LIN {X 0,Y 474.723,Z 291.355,A -85,B 0,C 180,E1 -7371.486,E2 -7371.486} C_VEL
LIN {X 0,Y 474.771,Z 291.342,A -85,B 0,C 180,E1 -7374.052,E2 -7374.052} C_VEL
LIN {X 0,Y 474.888,Z 291.331,A -85,B 0,C 180,E1 -7377.455,E2 -7377.455} C_VEL
LIN {X 0,Y 474.905,Z 291.328,A -85,B 0,C 180,E1 -7380,E2 -7380} C_VEL
LIN {X 0,Y 474.888,Z 291.326,A -85,B 0,C 180,E1 -7382.544,E2 -7382.544} C_VEL
LIN {X 0,Y 474.754,Z 291.35,A -85,B 0,C 180,E1 -7385.948,E2 -7385.948} C_VEL
LIN {X 0,Y 474.722,Z 291.348,A -85,B 0,C 180,E1 -7388.513,E2 -7388.513} C_VEL
LIN {X 0,Y 474.699,Z 291.357,A -85,B 0,C 180,E1 -7391.962,E2 -7391.962} C_VEL
LIN {X 0,Y 474.693,Z 291.35,A -85,B 0,C 180,E1 -7395.456,E2 -7395.456} C_VEL
LIN {X 0,Y 474.657,Z 291.355,A -85,B 0,C 180,E1 -7399.01,E2 -7399.01} C_VEL
LIN {X 0,Y 474.582,Z 291.365,A -85,B 0,C 180,E1 -7401.729,E2 -7401.729} C_VEL
LIN {X 0,Y 474.635,Z 291.365,A -85,B 0,C 180,E1 -7404.494,E2 -7404.494} C_VEL
LIN {X 0,Y 474.667,Z 291.353,A -85,B 0,C 180,E1 -7407.333,E2 -7407.333} C_VEL
LIN {X 0,Y 474.599,Z 291.366,A -85,B 0,C 180,E1 -7410.23,E2 -7410.23} C_VEL
LIN {X 0,Y 474.637,Z 291.358,A -85,B 0,C 180,E1 -7413.22,E2 -7413.22} C_VEL
LIN {X 0,Y 474.583,Z 291.367,A -85,B 0,C 180,E1 -7416.324,E2 -7416.324} C_VEL
LIN {X 0,Y 474.611,Z 291.36,A -85,B 0,C 180,E1 -7419.646,E2 -7419.646} C_VEL
LIN {X 0,Y 474.619,Z 291.36,A -85,B 0,C 180,E1 -7422.237,E2 -7422.237} C_VEL
LIN {X 0,Y 474.616,Z 291.363,A -85,B 0,C 180,E1 -7425.298,E2 -7425.298} C_VEL
LIN {X 0,Y 474.599,Z 291.362,A -85,B 0,C 180,E1 -7428.213,E2 -7428.213} C_VEL
LIN {X 0,Y 474.605,Z 291.364,A -85,B 0,C 180,E1 -7431.543,E2 -7431.543} C_VEL
LIN {X 0,Y 474.619,Z 291.361,A -85,B 0,C 180,E1 -7434.726,E2 -7434.726} C_VEL
LIN {X 0,Y 474.631,Z 291.36,A -85,B 0,C 180,E1 -7437.788,E2 -7437.788} C_VEL
LIN {X 0,Y 474.598,Z 291.364,A -85,B 0,C 180,E1 -7440.89,E2 -7440.89} C_VEL
LIN {X 0,Y 474.58,Z 291.37,A -85,B 0,C 180,E1 -7443.624,E2 -7443.624} C_VEL
LIN {X 0,Y 474.632,Z 291.357,A -85,B 0,C 180,E1 -7446.642,E2 -7446.642} C_VEL
LIN {X 0,Y 474.65,Z 291.358,A -85,B 0,C 180,E1 -7450.09,E2 -7450.09} C_VEL
LIN {X 0,Y 474.641,Z 291.361,A -85,B 0,C 180,E1 -7451.655,E2 -7451.655} C_VEL
LIN {X 0,Y 473.971,Z 291.446,A -85,B 0,C 180,E1 -7452.364,E2 -7452.364} C_VEL
LIN {X 0,Y 471.125,Z 291.8,A -85,B 0,C 180,E1 -7453.515,E2 -7453.515} C_VEL
LIN {X 0,Y 468.718,Z 292.097,A -85,B 0,C 180,E1 -7454.444,E2 -7454.444} C_VEL
LIN {X 0,Y 467.68,Z 292.225,A -85,B 0,C 180,E1 -7455.161,E2 -7455.161} C_VEL
LIN {X 0,Y 467.593,Z 292.236,A -85,B 0,C 180,E1 -7455.404,E2 -7455.404} C_VEL
LIN {X 0,Y 467.646,Z 292.237,A -85,B 0,C 180,E1 -7457.855,E2 -7457.855} C_VEL
LIN {X 0,Y 467.608,Z 292.446,A -85,B 0,C 180,E1 -7459.391,E2 -7459.391} C_VEL
LIN {X 0,Y 468.582,Z 298.825,A -85,B 0,C 180,E1 -7460.722,E2 -7460.722} C_VEL
LIN {X 0,Y 468.407,Z 309.742,A -85,B 0,C 180,E1 -7462.891,E2 -7462.891} C_VEL
LIN {X 0,Y 468.423,Z 311.097,A -85,B 0,C 180,E1 -7463.12,E2 -7463.12} C_VEL
LIN {X 0,Y 471.229,Z 325.691,A -85,B 0,C 180,E1 -7463.443,E2 -7463.443} C_VEL
LIN {X 0,Y 470.47,Z 418.633,A -85,B 0,C 180,E1 -7464.885,E2 -7464.885} C_VEL
LIN {X 0,Y 470.184,Z 432.296,A -85,B 0,C 180,E1 -7465.285,E2 -7465.285} C_VEL
LIN {X 0,Y 469.932,Z 444.537,A -85,B 0,C 180,E1 -7465.819,E2 -7465.819} C_VEL
LIN {X 0,Y 469.504,Z 455.551,A -85,B 0,C 180,E1 -7466.46,E2 -7466.46} C_VEL
LIN {X 0,Y 468.905,Z 467.03,A -85,B 0,C 180,E1 -7467.316,E2 -7467.316} C_VEL
LIN {X 0,Y 468.348,Z 477.362,A -85,B 0,C 180,E1 -7468.281,E2 -7468.281} C_VEL
LIN {X 0,Y 468.012,Z 486.652,A -85,B 0,C 180,E1 -7469.355,E2 -7469.355} C_VEL
LIN {X 0,Y 467.614,Z 495.635,A -85,B 0,C 180,E1 -7470.646,E2 -7470.646} C_VEL
LIN {X 0,Y 467.235,Z 502.903,A -85,B 0,C 180,E1 -7471.94,E2 -7471.94} C_VEL
LIN {X 0,Y 467.003,Z 509.572,A -85,B 0,C 180,E1 -7473.451,E2 -7473.451} C_VEL
LIN {X 0,Y 466.785,Z 513.994,A -85,B 0,C 180,E1 -7474.75,E2 -7474.75} C_VEL
LIN {X 0,Y 466.802,Z 517.34,A -85,B 0,C 180,E1 -7476.05,E2 -7476.05} C_VEL
LIN {X 0,Y 466.72,Z 519.012,A -85,B 0,C 180,E1 -7476.919,E2 -7476.919} C_VEL
LIN {X 0,Y 466.647,Z 520.285,A -85,B 0,C 180,E1 -7477.79,E2 -7477.79} C_VEL
LIN {X 0,Y 466.607,Z 521.161,A -85,B 0,C 180,E1 -7478.663,E2 -7478.663} C_VEL
LIN {X 0,Y 466.617,Z 521.635,A -85,B 0,C 180,E1 -7480.413,E2 -7480.413} C_VEL
LIN {X 0,Y 466.682,Z 520.881,A -85,B 0,C 180,E1 -7481.8,E2 -7481.8} C_VEL
LIN {X 0,Y 466.617,Z 519.325,A -85,B 0,C 180,E1 -7483.057,E2 -7483.057} C_VEL
LIN {X 0,Y 466.789,Z 516.721,A -85,B 0,C 180,E1 -7484.385,E2 -7484.385} C_VEL
LIN {X 0,Y 466.913,Z 513.055,A -85,B 0,C 180,E1 -7485.72,E2 -7485.72} C_VEL
LIN {X 0,Y 467.082,Z 508.207,A -85,B 0,C 180,E1 -7487.062,E2 -7487.062} C_VEL
LIN {X 0,Y 467.401,Z 502.021,A -85,B 0,C 180,E1 -7488.407,E2 -7488.407} C_VEL
LIN {X 0,Y 467.778,Z 494.252,A -85,B 0,C 180,E1 -7489.758,E2 -7489.758} C_VEL
LIN {X 0,Y 468.18,Z 486.207,A -85,B 0,C 180,E1 -7490.887,E2 -7490.887} C_VEL
LIN {X 0,Y 468.699,Z 476.286,A -85,B 0,C 180,E1 -7492.016,E2 -7492.016} C_VEL
LIN {X 0,Y 469.231,Z 465.174,A -85,B 0,C 180,E1 -7493.035,E2 -7493.035} C_VEL
LIN {X 0,Y 469.751,Z 454.217,A -85,B 0,C 180,E1 -7493.825,E2 -7493.825} C_VEL
LIN {X 0,Y 470.136,Z 442.648,A -85,B 0,C 180,E1 -7494.477,E2 -7494.477} C_VEL
LIN {X 0,Y 470.465,Z 429.508,A -85,B 0,C 180,E1 -7495.021,E2 -7495.021} C_VEL
LIN {X 0,Y 470.663,Z 418.167,A -85,B 0,C 180,E1 -7495.334,E2 -7495.334} C_VEL
LIN {X 0,Y 471.539,Z 325.876,A -85,B 0,C 180,E1 -7496.773,E2 -7496.773} C_VEL
LIN {X 0,Y 468.472,Z 310.826,A -85,B 0,C 180,E1 -7497.149,E2 -7497.149} C_VEL
LIN {X 0,Y 468.698,Z 298.454,A -85,B 0,C 180,E1 -7499.577,E2 -7499.577} C_VEL
LIN {X 0,Y 467.588,Z 292.242,A -85,B 0,C 180,E1 -7500.909,E2 -7500.909} C_VEL
LIN {X 0,Y 467.588,Z 292.243,A -85,B 0,C 180,E1 -7504.242,E2 -7504.242} C_VEL
LIN {X 0,Y 467.547,Z 292.238,A -85,B 0,C 180,E1 -7507.186,E2 -7507.186} C_VEL
LIN {X 0,Y 467.574,Z 292.243,A -85,B 0,C 180,E1 -7510.265,E2 -7510.265} C_VEL
LIN {X 0,Y 467.586,Z 292.242,A -85,B 0,C 180,E1 -7512.567,E2 -7512.567} C_VEL
LIN {X 0,Y 467.565,Z 292.243,A -85,B 0,C 180,E1 -7515.053,E2 -7515.053} C_VEL
LIN {X 0,Y 467.588,Z 292.236,A -85,B 0,C 180,E1 -7517.44,E2 -7517.44} C_VEL
LIN {X 0,Y 467.581,Z 292.243,A -85,B 0,C 180,E1 -7520.855,E2 -7520.855} C_VEL
LIN {X 0,Y 467.559,Z 292.238,A -85,B 0,C 180,E1 -7524.261,E2 -7524.261} C_VEL
LIN {X 0,Y 467.581,Z 292.238,A -85,B 0,C 180,E1 -7527.321,E2 -7527.321} C_VEL
LIN {X 0,Y 467.569,Z 292.237,A -85,B 0,C 180,E1 -7530.668,E2 -7530.668} C_VEL
LIN {X 0,Y 467.615,Z 292.234,A -85,B 0,C 180,E1 -7533.2,E2 -7533.2} C_VEL
LIN {X 0,Y 467.591,Z 292.23,A -85,B 0,C 180,E1 -7536.468,E2 -7536.468} C_VEL
LIN {X 0,Y 467.621,Z 292.23,A -85,B 0,C 180,E1 -7539.777,E2 -7539.777} C_VEL
LIN {X 0,Y 467.606,Z 292.233,A -85,B 0,C 180,E1 -7542.507,E2 -7542.507} C_VEL
LIN {X 0,Y 467.605,Z 292.233,A -85,B 0,C 180,E1 -7545.197,E2 -7545.197} C_VEL
LIN {X 0,Y 467.655,Z 292.23,A -85,B 0,C 180,E1 -7547.855,E2 -7547.855} C_VEL
LIN {X 0,Y 467.681,Z 292.227,A -85,B 0,C 180,E1 -7551.357,E2 -7551.357} C_VEL
LIN {X 0,Y 467.733,Z 292.222,A -85,B 0,C 180,E1 -7553.963,E2 -7553.963} C_VEL
LIN {X 0,Y 467.859,Z 292.202,A -85,B 0,C 180,E1 -7557.417,E2 -7557.417} C_VEL
LIN {X 0,Y 467.881,Z 292.205,A -85,B 0,C 180,E1 -7560,E2 -7560} C_VEL
LIN {X 0,Y 467.858,Z 292.201,A -85,B 0,C 180,E1 -7562.583,E2 -7562.583} C_VEL
LIN {X 0,Y 467.734,Z 292.222,A -85,B 0,C 180,E1 -7566.038,E2 -7566.038} C_VEL
LIN {X 0,Y 467.681,Z 292.227,A -85,B 0,C 180,E1 -7568.643,E2 -7568.643} C_VEL
LIN {X 0,Y 467.656,Z 292.227,A -85,B 0,C 180,E1 -7572.146,E2 -7572.146} C_VEL
LIN {X 0,Y 467.639,Z 292.226,A -85,B 0,C 180,E1 -7575.695,E2 -7575.695} C_VEL
LIN {X 0,Y 467.617,Z 292.236,A -85,B 0,C 180,E1 -7578.765,E2 -7578.765} C_VEL
LIN {X 0,Y 467.58,Z 292.237,A -85,B 0,C 180,E1 -7581.268,E2 -7581.268} C_VEL
LIN {X 0,Y 467.572,Z 292.236,A -85,B 0,C 180,E1 -7583.944,E2 -7583.944} C_VEL
LIN {X 0,Y 467.617,Z 292.24,A -85,B 0,C 180,E1 -7586.8,E2 -7586.8} C_VEL
LIN {X 0,Y 467.554,Z 292.24,A -85,B 0,C 180,E1 -7589.738,E2 -7589.738} C_VEL
LIN {X 0,Y 467.584,Z 292.239,A -85,B 0,C 180,E1 -7592.759,E2 -7592.759} C_VEL
LIN {X 0,Y 467.554,Z 292.238,A -85,B 0,C 180,E1 -7595.89,E2 -7595.89} C_VEL
LIN {X 0,Y 467.577,Z 292.238,A -85,B 0,C 180,E1 -7599.146,E2 -7599.146} C_VEL
LIN {X 0,Y 467.588,Z 292.235,A -85,B 0,C 180,E1 -7602.567,E2 -7602.567} C_VEL
LIN {X 0,Y 467.567,Z 292.241,A -85,B 0,C 180,E1 -7605.053,E2 -7605.053} C_VEL
LIN {X 0,Y 467.591,Z 292.242,A -85,B 0,C 180,E1 -7607.44,E2 -7607.44} C_VEL
LIN {X 0,Y 467.562,Z 292.24,A -85,B 0,C 180,E1 -7610.853,E2 -7610.853} C_VEL
LIN {X 0,Y 467.562,Z 292.242,A -85,B 0,C 180,E1 -7614.261,E2 -7614.261} C_VEL
LIN {X 0,Y 467.584,Z 292.241,A -85,B 0,C 180,E1 -7617.321,E2 -7617.321} C_VEL
LIN {X 0,Y 467.572,Z 292.241,A -85,B 0,C 180,E1 -7620.668,E2 -7620.668} C_VEL
LIN {X 0,Y 467.656,Z 292.33,A -85,B 0,C 180,E1 -7623.803,E2 -7623.803} C_VEL
LIN {X 0,Y 469.784,Z 303.007,A -85,B 0,C 180,E1 -7625.863,E2 -7625.863} C_VEL
LIN {X 0,Y 469.808,Z 309.972,A -85,B 0,C 180,E1 -7627.111,E2 -7627.111} C_VEL
LIN {X 0,Y 468.912,Z 329.539,A -85,B 0,C 180,E1 -7630.52,E2 -7630.52} C_VEL
LIN {X 0,Y 468.369,Z 343.57,A -85,B 0,C 180,E1 -7632.905,E2 -7632.905} C_VEL
LIN {X 0,Y 471.319,Z 363.38,A -85,B 0,C 180,E1 -7633.336,E2 -7633.336} C_VEL
LIN {X 0,Y 470.655,Z 451.588,A -85,B 0,C 180,E1 -7634.713,E2 -7634.713} C_VEL
LIN {X 0,Y 470.26,Z 464.156,A -85,B 0,C 180,E1 -7635.06,E2 -7635.06} C_VEL
LIN {X 0,Y 469.811,Z 477.1,A -85,B 0,C 180,E1 -7635.599,E2 -7635.599} C_VEL
LIN {X 0,Y 469.33,Z 488.59,A -85,B 0,C 180,E1 -7636.248,E2 -7636.248} C_VEL
LIN {X 0,Y 468.867,Z 499.09,A -85,B 0,C 180,E1 -7637.006,E2 -7637.006} C_VEL
LIN {X 0,Y 468.361,Z 509.888,A -85,B 0,C 180,E1 -7637.983,E2 -7637.983} C_VEL
LIN {X 0,Y 467.794,Z 520.504,A -85,B 0,C 180,E1 -7639.176,E2 -7639.176} C_VEL
LIN {X 0,Y 467.345,Z 529.701,A -85,B 0,C 180,E1 -7640.478,E2 -7640.478} C_VEL
LIN {X 0,Y 467.066,Z 537.117,A -85,B 0,C 180,E1 -7641.781,E2 -7641.781} C_VEL
LIN {X 0,Y 466.851,Z 543.077,A -85,B 0,C 180,E1 -7643.083,E2 -7643.083} C_VEL
LIN {X 0,Y 466.761,Z 547.79,A -85,B 0,C 180,E1 -7644.383,E2 -7644.383} C_VEL
LIN {X 0,Y 466.647,Z 551.39,A -85,B 0,C 180,E1 -7645.681,E2 -7645.681} C_VEL
LIN {X 0,Y 466.69,Z 553.248,A -85,B 0,C 180,E1 -7646.546,E2 -7646.546} C_VEL
LIN {X 0,Y 466.662,Z 554.64,A -85,B 0,C 180,E1 -7647.41,E2 -7647.41} C_VEL
LIN {X 0,Y 466.619,Z 556.241,A -85,B 0,C 180,E1 -7649.137,E2 -7649.137} C_VEL
LIN {X 0,Y 466.601,Z 556.45,A -85,B 0,C 180,E1 -7650,E2 -7650} C_VEL
LIN {X 0,Y 466.619,Z 556.228,A -85,B 0,C 180,E1 -7650.863,E2 -7650.863} C_VEL
LIN {X 0,Y 466.662,Z 554.614,A -85,B 0,C 180,E1 -7652.589,E2 -7652.589} C_VEL
LIN {X 0,Y 466.69,Z 553.205,A -85,B 0,C 180,E1 -7653.453,E2 -7653.453} C_VEL
LIN {X 0,Y 466.689,Z 550.247,A -85,B 0,C 180,E1 -7654.751,E2 -7654.751} C_VEL
LIN {X 0,Y 466.75,Z 546.241,A -85,B 0,C 180,E1 -7656.05,E2 -7656.05} C_VEL
LIN {X 0,Y 466.925,Z 540.074,A -85,B 0,C 180,E1 -7657.568,E2 -7657.568} C_VEL
LIN {X 0,Y 467.165,Z 533.341,A -85,B 0,C 180,E1 -7658.87,E2 -7658.87} C_VEL
LIN {X 0,Y 467.506,Z 524.984,A -85,B 0,C 180,E1 -7660.174,E2 -7660.174} C_VEL
LIN {X 0,Y 467.972,Z 516.394,A -85,B 0,C 180,E1 -7661.258,E2 -7661.258} C_VEL
LIN {X 0,Y 468.463,Z 506.224,A -85,B 0,C 180,E1 -7662.302,E2 -7662.302} C_VEL
LIN {X 0,Y 468.881,Z 495.252,A -85,B 0,C 180,E1 -7663.213,E2 -7663.213} C_VEL
LIN {X 0,Y 469.403,Z 483.651,A -85,B 0,C 180,E1 -7663.97,E2 -7663.97} C_VEL
LIN {X 0,Y 469.866,Z 471.593,A -85,B 0,C 180,E1 -7664.564,E2 -7664.564} C_VEL
LIN {X 0,Y 470.219,Z 458.518,A -85,B 0,C 180,E1 -7665.024,E2 -7665.024} C_VEL
LIN {X 0,Y 470.502,Z 446.174,A -85,B 0,C 180,E1 -7665.291,E2 -7665.291} C_VEL
LIN {X 0,Y 471.087,Z 362.941,A -85,B 0,C 180,E1 -7666.562,E2 -7666.562} C_VEL
LIN {X 0,Y 468.226,Z 343.525,A -85,B 0,C 180,E1 -7666.969,E2 -7666.969} C_VEL
LIN {X 0,Y 468.921,Z 326.108,A -85,B 0,C 180,E1 -7669.935,E2 -7669.935} C_VEL
LIN {X 0,Y 469.726,Z 306.247,A -85,B 0,C 180,E1 -7673.358,E2 -7673.358} C_VEL
LIN {X 0,Y 469.556,Z 302.21,A -85,B 0,C 180,E1 -7674.075,E2 -7674.075} C_VEL
LIN {X 0,Y 467.65,Z 292.236,A -85,B 0,C 180,E1 -7675.957,E2 -7675.957} C_VEL
LIN {X 0,Y 467.577,Z 292.241,A -85,B 0,C 180,E1 -7678.749,E2 -7678.749} C_VEL
LIN {X 0,Y 467.583,Z 292.239,A -85,B 0,C 180,E1 -7681.739,E2 -7681.739} C_VEL
LIN {X 0,Y 467.563,Z 292.239,A -85,B 0,C 180,E1 -7684.832,E2 -7684.832} C_VEL
LIN {X 0,Y 467.564,Z 292.243,A -85,B 0,C 180,E1 -7688.044,E2 -7688.044} C_VEL
LIN {X 0,Y 467.577,Z 292.236,A -85,B 0,C 180,E1 -7691.276,E2 -7691.276} C_VEL
LIN {X 0,Y 467.55,Z 292.241,A -85,B 0,C 180,E1 -7693.82,E2 -7693.82} C_VEL
LIN {X 0,Y 467.552,Z 292.244,A -85,B 0,C 180,E1 -7696.255,E2 -7696.255} C_VEL
LIN {X 0,Y 467.576,Z 292.243,A -85,B 0,C 180,E1 -7698.723,E2 -7698.723} C_VEL
LIN {X 0,Y 467.562,Z 292.239,A -85,B 0,C 180,E1 -7701.955,E2 -7701.955} C_VEL
LIN {X 0,Y 467.561,Z 292.242,A -85,B 0,C 180,E1 -7705.167,E2 -7705.167} C_VEL
LIN {X 0,Y 467.579,Z 292.237,A -85,B 0,C 180,E1 -7708.259,E2 -7708.259} C_VEL
LIN {X 0,Y 467.573,Z 292.241,A -85,B 0,C 180,E1 -7711.25,E2 -7711.25} C_VEL
LIN {X 0,Y 467.606,Z 292.233,A -85,B 0,C 180,E1 -7714.16,E2 -7714.16} C_VEL
LIN {X 0,Y 467.573,Z 292.244,A -85,B 0,C 180,E1 -7716.995,E2 -7716.995} C_VEL
LIN {X 0,Y 467.618,Z 292.232,A -85,B 0,C 180,E1 -7719.777,E2 -7719.777} C_VEL
LIN {X 0,Y 467.604,Z 292.233,A -85,B 0,C 180,E1 -7722.506,E2 -7722.506} C_VEL
LIN {X 0,Y 467.605,Z 292.24,A -85,B 0,C 180,E1 -7725.196,E2 -7725.196} C_VEL
LIN {X 0,Y 467.651,Z 292.23,A -85,B 0,C 180,E1 -7727.854,E2 -7727.854} C_VEL
LIN {X 0,Y 467.677,Z 292.231,A -85,B 0,C 180,E1 -7731.357,E2 -7731.357} C_VEL
LIN {X 0,Y 467.735,Z 292.22,A -85,B 0,C 180,E1 -7733.962,E2 -7733.962} C_VEL
LIN {X 0,Y 467.853,Z 292.207,A -85,B 0,C 180,E1 -7737.417,E2 -7737.417} C_VEL
LIN {X 0,Y 467.875,Z 292.204,A -85,B 0,C 180,E1 -7740,E2 -7740} C_VEL
LIN {X 0,Y 467.854,Z 292.202,A -85,B 0,C 180,E1 -7742.583,E2 -7742.583} C_VEL
LIN {X 0,Y 467.716,Z 292.226,A -85,B 0,C 180,E1 -7746.038,E2 -7746.038} C_VEL
LIN {X 0,Y 467.676,Z 292.225,A -85,B 0,C 180,E1 -7748.643,E2 -7748.643} C_VEL
LIN {X 0,Y 467.65,Z 292.235,A -85,B 0,C 180,E1 -7752.145,E2 -7752.145} C_VEL
LIN {X 0,Y 467.633,Z 292.232,A -85,B 0,C 180,E1 -7755.695,E2 -7755.695} C_VEL
LIN {X 0,Y 467.616,Z 292.231,A -85,B 0,C 180,E1 -7759.308,E2 -7759.308} C_VEL
LIN {X 0,Y 467.529,Z 292.247,A -85,B 0,C 180,E1 -7762.074,E2 -7762.074} C_VEL
LIN {X 0,Y 467.58,Z 292.238,A -85,B 0,C 180,E1 -7764.889,E2 -7764.889} C_VEL
LIN {X 0,Y 467.61,Z 292.233,A -85,B 0,C 180,E1 -7767.77,E2 -7767.77} C_VEL
LIN {X 0,Y 467.562,Z 292.241,A -85,B 0,C 180,E1 -7771.045,E2 -7771.045} C_VEL
LIN {X 0,Y 467.583,Z 292.239,A -85,B 0,C 180,E1 -7774.242,E2 -7774.242} C_VEL
LIN {X 0,Y 467.542,Z 292.243,A -85,B 0,C 180,E1 -7777.186,E2 -7777.186} C_VEL
LIN {X 0,Y 467.569,Z 292.239,A -85,B 0,C 180,E1 -7780.265,E2 -7780.265} C_VEL
LIN {X 0,Y 467.582,Z 292.24,A -85,B 0,C 180,E1 -7782.567,E2 -7782.567} C_VEL
LIN {X 0,Y 467.566,Z 292.245,A -85,B 0,C 180,E1 -7785.053,E2 -7785.053} C_VEL
LIN {X 0,Y 467.56,Z 292.242,A -85,B 0,C 180,E1 -7788.726,E2 -7788.726} C_VEL
LIN {X 0,Y 467.559,Z 292.239,A -85,B 0,C 180,E1 -7791.956,E2 -7791.956} C_VEL
LIN {X 0,Y 467.555,Z 292.247,A -85,B 0,C 180,E1 -7795.167,E2 -7795.167} C_VEL
LIN {X 0,Y 467.578,Z 292.236,A -85,B 0,C 180,E1 -7798.26,E2 -7798.26} C_VEL
LIN {X 0,Y 467.544,Z 292.247,A -85,B 0,C 180,E1 -7801.249,E2 -7801.249} C_VEL
LIN {X 0,Y 467.573,Z 292.237,A -85,B 0,C 180,E1 -7804.402,E2 -7804.402} C_VEL
LIN {X 0,Y 467.574,Z 292.238,A -85,B 0,C 180,E1 -7806.996,E2 -7806.996} C_VEL
LIN {X 0,Y 467.619,Z 292.238,A -85,B 0,C 180,E1 -7809.778,E2 -7809.778} C_VEL
LIN {X 0,Y 467.589,Z 292.235,A -85,B 0,C 180,E1 -7812.506,E2 -7812.506} C_VEL
LIN {X 0,Y 467.602,Z 292.235,A -85,B 0,C 180,E1 -7815.197,E2 -7815.197} C_VEL
LIN {X 0,Y 467.593,Z 292.236,A -85,B 0,C 180,E1 -7815.404,E2 -7815.404} C_VEL
LIN {X 0,Y 466.917,Z 292.326,A -85,B 0,C 180,E1 -7815.883,E2 -7815.883} C_VEL
LIN {X 0,Y 464.102,Z 292.676,A -85,B 0,C 180,E1 -7816.634,E2 -7816.634} C_VEL
LIN {X 0,Y 461.27,Z 293.03,A -85,B 0,C 180,E1 -7817.393,E2 -7817.393} C_VEL
LIN {X 0,Y 460.588,Z 293.114,A -85,B 0,C 180,E1 -7817.883,E2 -7817.883} C_VEL
LIN {X 0,Y 460.589,Z 293.244,A -85,B 0,C 180,E1 -7819.227,E2 -7819.227} C_VEL
LIN {X 0,Y 461.59,Z 299.658,A -85,B 0,C 180,E1 -7820.58,E2 -7820.58} C_VEL
LIN {X 0,Y 461.453,Z 308.434,A -85,B 0,C 180,E1 -7822.344,E2 -7822.344} C_VEL
LIN {X 0,Y 461.421,Z 311.167,A -85,B 0,C 180,E1 -7822.879,E2 -7822.879} C_VEL
LIN {X 0,Y 464.42,Z 327.318,A -85,B 0,C 180,E1 -7823.238,E2 -7823.238} C_VEL
LIN {X 0,Y 463.599,Z 418.669,A -85,B 0,C 180,E1 -7824.673,E2 -7824.673} C_VEL
LIN {X 0,Y 463.295,Z 432.41,A -85,B 0,C 180,E1 -7825.078,E2 -7825.078} C_VEL
LIN {X 0,Y 463.005,Z 445.221,A -85,B 0,C 180,E1 -7825.648,E2 -7825.648} C_VEL
LIN {X 0,Y 462.512,Z 457.693,A -85,B 0,C 180,E1 -7826.407,E2 -7826.407} C_VEL
LIN {X 0,Y 461.896,Z 468.832,A -85,B 0,C 180,E1 -7827.275,E2 -7827.275} C_VEL
LIN {X 0,Y 461.358,Z 478.868,A -85,B 0,C 180,E1 -7828.254,E2 -7828.254} C_VEL
LIN {X 0,Y 460.975,Z 487.898,A -85,B 0,C 180,E1 -7829.345,E2 -7829.345} C_VEL
LIN {X 0,Y 460.554,Z 496.719,A -85,B 0,C 180,E1 -7830.656,E2 -7830.656} C_VEL
LIN {X 0,Y 460.165,Z 503.844,A -85,B 0,C 180,E1 -7831.97,E2 -7831.97} C_VEL
LIN {X 0,Y 459.964,Z 508.65,A -85,B 0,C 180,E1 -7833.066,E2 -7833.066} C_VEL
LIN {X 0,Y 459.754,Z 513.335,A -85,B 0,C 180,E1 -7834.384,E2 -7834.384} C_VEL
LIN {X 0,Y 459.738,Z 516.914,A -85,B 0,C 180,E1 -7835.703,E2 -7835.703} C_VEL
LIN {X 0,Y 459.625,Z 519.502,A -85,B 0,C 180,E1 -7837.027,E2 -7837.027} C_VEL
LIN {X 0,Y 459.542,Z 520.725,A -85,B 0,C 180,E1 -7837.912,E2 -7837.912} C_VEL
LIN {X 0,Y 459.503,Z 521.51,A -85,B 0,C 180,E1 -7838.798,E2 -7838.798} C_VEL
LIN {X 0,Y 459.536,Z 521.875,A -85,B 0,C 180,E1 -7840.575,E2 -7840.575} C_VEL
LIN {X 0,Y 459.588,Z 521.142,A -85,B 0,C 180,E1 -7841.852,E2 -7841.852} C_VEL
LIN {X 0,Y 459.558,Z 519.362,A -85,B 0,C 180,E1 -7843.262,E2 -7843.262} C_VEL
LIN {X 0,Y 459.721,Z 516.652,A -85,B 0,C 180,E1 -7844.611,E2 -7844.611} C_VEL
LIN {X 0,Y 459.879,Z 512.873,A -85,B 0,C 180,E1 -7845.967,E2 -7845.967} C_VEL
LIN {X 0,Y 460.074,Z 507.903,A -85,B 0,C 180,E1 -7847.33,E2 -7847.33} C_VEL
LIN {X 0,Y 460.429,Z 501.585,A -85,B 0,C 180,E1 -7848.696,E2 -7848.696} C_VEL
LIN {X 0,Y 460.779,Z 495.065,A -85,B 0,C 180,E1 -7849.838,E2 -7849.838} C_VEL
LIN {X 0,Y 461.194,Z 487.167,A -85,B 0,C 180,E1 -7850.984,E2 -7850.984} C_VEL
LIN {X 0,Y 461.761,Z 477.198,A -85,B 0,C 180,E1 -7852.154,E2 -7852.154} C_VEL
LIN {X 0,Y 462.313,Z 466.507,A -85,B 0,C 180,E1 -7853.163,E2 -7853.163} C_VEL
LIN {X 0,Y 462.865,Z 455.89,A -85,B 0,C 180,E1 -7853.964,E2 -7853.964} C_VEL
LIN {X 0,Y 463.265,Z 444.078,A -85,B 0,C 180,E1 -7854.662,E2 -7854.662} C_VEL
LIN {X 0,Y 463.654,Z 430.754,A -85,B 0,C 180,E1 -7855.234,E2 -7855.234} C_VEL
LIN {X 0,Y 463.868,Z 418.708,A -85,B 0,C 180,E1 -7855.582,E2 -7855.582} C_VEL
LIN {X 0,Y 464.792,Z 326.54,A -85,B 0,C 180,E1 -7857.043,E2 -7857.043} C_VEL
LIN {X 0,Y 461.586,Z 311.005,A -85,B 0,C 180,E1 -7857.455,E2 -7857.455} C_VEL
LIN {X 0,Y 461.827,Z 300.836,A -85,B 0,C 180,E1 -7859.472,E2 -7859.472} C_VEL
LIN {X 0,Y 460.919,Z 294.908,A -85,B 0,C 180,E1 -7860.717,E2 -7860.717} C_VEL
LIN {X 0,Y 460.543,Z 293.12,A -85,B 0,C 180,E1 -7861.127,E2 -7861.127} C_VEL
LIN {X 0,Y 460.531,Z 293.123,A -85,B 0,C 180,E1 -7864.506,E2 -7864.506} C_VEL
LIN {X 0,Y 460.5,Z 293.115,A -85,B 0,C 180,E1 -7867.623,E2 -7867.623} C_VEL
LIN {X 0,Y 460.538,Z 293.119,A -85,B 0,C 180,E1 -7870.269,E2 -7870.269} C_VEL
LIN {X 0,Y 460.497,Z 293.12,A -85,B 0,C 180,E1 -7873.376,E2 -7873.376} C_VEL
LIN {X 0,Y 460.498,Z 293.126,A -85,B 0,C 180,E1 -7876.625,E2 -7876.625} C_VEL
LIN {X 0,Y 460.541,Z 293.113,A -85,B 0,C 180,E1 -7879.731,E2 -7879.731} C_VEL
LIN {X 0,Y 460.498,Z 293.121,A -85,B 0,C 180,E1 -7882.524,E2 -7882.524} C_VEL
LIN {X 0,Y 460.545,Z 293.111,A -85,B 0,C 180,E1 -7885.624,E2 -7885.624} C_VEL
LIN {X 0,Y 460.536,Z 293.115,A -85,B 0,C 180,E1 -7888.745,E2 -7888.745} C_VEL
LIN {X 0,Y 460.58,Z 293.104,A -85,B 0,C 180,E1 -7892.254,E2 -7892.254} C_VEL
LIN {X 0,Y 460.546,Z 293.112,A -85,B 0,C 180,E1 -7894.705,E2 -7894.705} C_VEL
LIN {X 0,Y 460.51,Z 293.121,A -85,B 0,C 180,E1 -7897.571,E2 -7897.571} C_VEL
LIN {X 0,Y 460.568,Z 293.105,A -85,B 0,C 180,E1 -7900.385,E2 -7900.385} C_VEL
LIN {X 0,Y 460.563,Z 293.114,A -85,B 0,C 180,E1 -7903.146,E2 -7903.146} C_VEL
LIN {X 0,Y 460.554,Z 293.117,A -85,B 0,C 180,E1 -7905.868,E2 -7905.868} C_VEL
LIN {X 0,Y 460.61,Z 293.102,A -85,B 0,C 180,E1 -7908.559,E2 -7908.559} C_VEL
LIN {X 0,Y 460.695,Z 293.096,A -85,B 0,C 180,E1 -7912.109,E2 -7912.109} C_VEL
LIN {X 0,Y 460.692,Z 293.093,A -85,B 0,C 180,E1 -7914.748,E2 -7914.748} C_VEL
LIN {X 0,Y 460.8,Z 293.081,A -85,B 0,C 180,E1 -7917.378,E2 -7917.378} C_VEL
LIN {X 0,Y 460.852,Z 293.081,A -85,B 0,C 180,E1 -7920,E2 -7920} C_VEL
LIN {X 0,Y 460.799,Z 293.079,A -85,B 0,C 180,E1 -7922.623,E2 -7922.623} C_VEL
LIN {X 0,Y 460.7,Z 293.098,A -85,B 0,C 180,E1 -7926.13,E2 -7926.13} C_VEL
LIN {X 0,Y 460.628,Z 293.104,A -85,B 0,C 180,E1 -7928.776,E2 -7928.776} C_VEL
LIN {X 0,Y 460.613,Z 293.107,A -85,B 0,C 180,E1 -7932.445,E2 -7932.445} C_VEL
LIN {X 0,Y 460.6,Z 293.105,A -85,B 0,C 180,E1 -7935.998,E2 -7935.998} C_VEL
LIN {X 0,Y 460.571,Z 293.112,A -85,B 0,C 180,E1 -7938.902,E2 -7938.902} C_VEL
LIN {X 0,Y 460.516,Z 293.116,A -85,B 0,C 180,E1 -7941.486,E2 -7941.486} C_VEL
LIN {X 0,Y 460.542,Z 293.115,A -85,B 0,C 180,E1 -7944.333,E2 -7944.333} C_VEL
LIN {X 0,Y 460.573,Z 293.112,A -85,B 0,C 180,E1 -7947.244,E2 -7947.244} C_VEL
LIN {X 0,Y 460.511,Z 293.118,A -85,B 0,C 180,E1 -7950.24,E2 -7950.24} C_VEL
LIN {X 0,Y 460.529,Z 293.12,A -85,B 0,C 180,E1 -7953.325,E2 -7953.325} C_VEL
LIN {X 0,Y 460.477,Z 293.12,A -85,B 0,C 180,E1 -7956.53,E2 -7956.53} C_VEL
LIN {X 0,Y 460.528,Z 293.106,A -85,B 0,C 180,E1 -7959.863,E2 -7959.863} C_VEL
LIN {X 0,Y 460.514,Z 293.119,A -85,B 0,C 180,E1 -7962.901,E2 -7962.901} C_VEL
LIN {X 0,Y 460.508,Z 293.121,A -85,B 0,C 180,E1 -7965.831,E2 -7965.831} C_VEL
LIN {X 0,Y 460.532,Z 293.117,A -85,B 0,C 180,E1 -7968.989,E2 -7968.989} C_VEL
LIN {X 0,Y 460.52,Z 293.12,A -85,B 0,C 180,E1 -7971.266,E2 -7971.266} C_VEL
LIN {X 0,Y 460.512,Z 293.119,A -85,B 0,C 180,E1 -7974.555,E2 -7974.555} C_VEL
LIN {X 0,Y 460.534,Z 293.119,A -85,B 0,C 180,E1 -7977.716,E2 -7977.716} C_VEL
LIN {X 0,Y 460.542,Z 293.117,A -85,B 0,C 180,E1 -7980.769,E2 -7980.769} C_VEL
LIN {X 0,Y 460.623,Z 293.244,A -85,B 0,C 180,E1 -7983.555,E2 -7983.555} C_VEL
LIN {X 0,Y 462.914,Z 304.669,A -85,B 0,C 180,E1 -7985.8,E2 -7985.8} C_VEL
LIN {X 0,Y 462.899,Z 311.186,A -85,B 0,C 180,E1 -7986.986,E2 -7986.986} C_VEL
LIN {X 0,Y 461.933,Z 330.734,A -85,B 0,C 180,E1 -7990.445,E2 -7990.445} C_VEL
LIN {X 0,Y 461.361,Z 343.102,A -85,B 0,C 180,E1 -7992.603,E2 -7992.603} C_VEL
LIN {X 0,Y 464.573,Z 363.589,A -85,B 0,C 180,E1 -7993.069,E2 -7993.069} C_VEL
LIN {X 0,Y 463.847,Z 452.275,A -85,B 0,C 180,E1 -7994.483,E2 -7994.483} C_VEL
LIN {X 0,Y 463.435,Z 464.514,A -85,B 0,C 180,E1 -7994.835,E2 -7994.835} C_VEL
LIN {X 0,Y 462.958,Z 477.288,A -85,B 0,C 180,E1 -7995.382,E2 -7995.382} C_VEL
LIN {X 0,Y 462.451,Z 488.656,A -85,B 0,C 180,E1 -7996.039,E2 -7996.039} C_VEL
LIN {X 0,Y 461.829,Z 500.689,A -85,B 0,C 180,E1 -7996.945,E2 -7996.945} C_VEL
LIN {X 0,Y 461.344,Z 510.89,A -85,B 0,C 180,E1 -7997.909,E2 -7997.909} C_VEL
LIN {X 0,Y 460.798,Z 520.392,A -85,B 0,C 180,E1 -7999.009,E2 -7999.009} C_VEL
LIN {X 0,Y 460.331,Z 529.551,A -85,B 0,C 180,E1 -8000.332,E2 -8000.332} C_VEL
LIN {X 0,Y 460.002,Z 536.941,A -85,B 0,C 180,E1 -8001.654,E2 -8001.654} C_VEL
LIN {X 0,Y 459.77,Z 542.881,A -85,B 0,C 180,E1 -8002.976,E2 -8002.976} C_VEL
LIN {X 0,Y 459.658,Z 547.577,A -85,B 0,C 180,E1 -8004.296,E2 -8004.296} C_VEL
LIN {X 0,Y 459.565,Z 551.163,A -85,B 0,C 180,E1 -8005.614,E2 -8005.614} C_VEL
LIN {X 0,Y 459.585,Z 553.01,A -85,B 0,C 180,E1 -8006.493,E2 -8006.493} C_VEL
LIN {X 0,Y 459.584,Z 554.395,A -85,B 0,C 180,E1 -8007.37,E2 -8007.37} C_VEL
LIN {X 0,Y 459.523,Z 555.985,A -85,B 0,C 180,E1 -8009.123,E2 -8009.123} C_VEL
LIN {X 0,Y 459.532,Z 556.186,A -85,B 0,C 180,E1 -8010,E2 -8010} C_VEL
LIN {X 0,Y 459.552,Z 555.956,A -85,B 0,C 180,E1 -8010.876,E2 -8010.876} C_VEL
LIN {X 0,Y 459.584,Z 554.33,A -85,B 0,C 180,E1 -8012.629,E2 -8012.629} C_VEL
LIN {X 0,Y 459.586,Z 552.91,A -85,B 0,C 180,E1 -8013.507,E2 -8013.507} C_VEL
LIN {X 0,Y 459.617,Z 549.942,A -85,B 0,C 180,E1 -8014.824,E2 -8014.824} C_VEL
LIN {X 0,Y 459.714,Z 544.872,A -85,B 0,C 180,E1 -8016.43,E2 -8016.43} C_VEL
LIN {X 0,Y 459.892,Z 538.713,A -85,B 0,C 180,E1 -8017.905,E2 -8017.905} C_VEL
LIN {X 0,Y 460.187,Z 531.728,A -85,B 0,C 180,E1 -8019.227,E2 -8019.227} C_VEL
LIN {X 0,Y 460.57,Z 522.964,A -85,B 0,C 180,E1 -8020.551,E2 -8020.551} C_VEL
LIN {X 0,Y 461.068,Z 513.99,A -85,B 0,C 180,E1 -8021.652,E2 -8021.652} C_VEL
LIN {X 0,Y 461.58,Z 503.142,A -85,B 0,C 180,E1 -8022.732,E2 -8022.732} C_VEL
LIN {X 0,Y 462.107,Z 491.641,A -85,B 0,C 180,E1 -8023.634,E2 -8023.634} C_VEL
LIN {X 0,Y 462.647,Z 479.007,A -85,B 0,C 180,E1 -8024.403,E2 -8024.403} C_VEL
LIN {X 0,Y 463.144,Z 465.986,A -85,B 0,C 180,E1 -8024.977,E2 -8024.977} C_VEL
LIN {X 0,Y 463.517,Z 453.152,A -85,B 0,C 180,E1 -8025.359,E2 -8025.359} C_VEL
LIN {X 0,Y 463.877,Z 416.778,A -85,B 0,C 180,E1 -8025.951,E2 -8025.951} C_VEL
LIN {X 0,Y 464.092,Z 362.235,A -85,B 0,C 180,E1 -8026.802,E2 -8026.802} C_VEL
LIN {X 0,Y 461.244,Z 343.19,A -85,B 0,C 180,E1 -8027.221,E2 -8027.221} C_VEL
LIN {X 0,Y 461.908,Z 327.003,A -85,B 0,C 180,E1 -8030.019,E2 -8030.019} C_VEL
LIN {X 0,Y 462.735,Z 308.459,A -85,B 0,C 180,E1 -8033.258,E2 -8033.258} C_VEL
LIN {X 0,Y 462.74,Z 304.459,A -85,B 0,C 180,E1 -8033.97,E2 -8033.97} C_VEL
LIN {X 0,Y 460.589,Z 293.115,A -85,B 0,C 180,E1 -8036.136,E2 -8036.136} C_VEL
LIN {X 0,Y 460.54,Z 293.117,A -85,B 0,C 180,E1 -8039.23,E2 -8039.23} C_VEL
LIN {X 0,Y 460.531,Z 293.121,A -85,B 0,C 180,E1 -8042.284,E2 -8042.284} C_VEL
LIN {X 0,Y 460.509,Z 293.117,A -85,B 0,C 180,E1 -8045.445,E2 -8045.445} C_VEL
LIN {X 0,Y 460.533,Z 293.115,A -85,B 0,C 180,E1 -8048.895,E2 -8048.895} C_VEL
LIN {X 0,Y 460.521,Z 293.12,A -85,B 0,C 180,E1 -8052.181,E2 -8052.181} C_VEL
LIN {X 0,Y 460.511,Z 293.116,A -85,B 0,C 180,E1 -8055.41,E2 -8055.41} C_VEL
LIN {X 0,Y 460.53,Z 293.12,A -85,B 0,C 180,E1 -8058.397,E2 -8058.397} C_VEL
LIN {X 0,Y 460.523,Z 293.116,A -85,B 0,C 180,E1 -8061.266,E2 -8061.266} C_VEL
LIN {X 0,Y 460.507,Z 293.123,A -85,B 0,C 180,E1 -8064.554,E2 -8064.554} C_VEL
LIN {X 0,Y 460.528,Z 293.114,A -85,B 0,C 180,E1 -8067.715,E2 -8067.715} C_VEL
LIN {X 0,Y 460.536,Z 293.12,A -85,B 0,C 180,E1 -8070.769,E2 -8070.769} C_VEL
LIN {X 0,Y 460.559,Z 293.111,A -85,B 0,C 180,E1 -8073.734,E2 -8073.734} C_VEL
LIN {X 0,Y 460.542,Z 293.115,A -85,B 0,C 180,E1 -8076.624,E2 -8076.624} C_VEL
LIN {X 0,Y 460.547,Z 293.117,A -85,B 0,C 180,E1 -8079.452,E2 -8079.452} C_VEL
LIN {X 0,Y 460.554,Z 293.111,A -85,B 0,C 180,E1 -8082.23,E2 -8082.23} C_VEL
LIN {X 0,Y 460.563,Z 293.114,A -85,B 0,C 180,E1 -8084.965,E2 -8084.965} C_VEL
LIN {X 0,Y 460.606,Z 293.105,A -85,B 0,C 180,E1 -8088.559,E2 -8088.559} C_VEL
LIN {X 0,Y 460.69,Z 293.096,A -85,B 0,C 180,E1 -8092.108,E2 -8092.108} C_VEL
LIN {X 0,Y 460.69,Z 293.094,A -85,B 0,C 180,E1 -8094.748,E2 -8094.748} C_VEL
LIN {X 0,Y 460.794,Z 293.086,A -85,B 0,C 180,E1 -8097.377,E2 -8097.377} C_VEL
LIN {X 0,Y 460.846,Z 293.079,A -85,B 0,C 180,E1 -8100,E2 -8100} C_VEL
LIN {X 0,Y 460.795,Z 293.081,A -85,B 0,C 180,E1 -8102.622,E2 -8102.622} C_VEL
LIN {X 0,Y 460.68,Z 293.101,A -85,B 0,C 180,E1 -8106.13,E2 -8106.13} C_VEL
LIN {X 0,Y 460.623,Z 293.103,A -85,B 0,C 180,E1 -8108.776,E2 -8108.776} C_VEL
LIN {X 0,Y 460.608,Z 293.108,A -85,B 0,C 180,E1 -8112.445,E2 -8112.445} C_VEL
LIN {X 0,Y 460.595,Z 293.112,A -85,B 0,C 180,E1 -8115.998,E2 -8115.998} C_VEL
LIN {X 0,Y 460.562,Z 293.111,A -85,B 0,C 180,E1 -8119.616,E2 -8119.616} C_VEL
LIN {X 0,Y 460.505,Z 293.125,A -85,B 0,C 180,E1 -8122.429,E2 -8122.429} C_VEL
LIN {X 0,Y 460.543,Z 293.114,A -85,B 0,C 180,E1 -8125.797,E2 -8125.797} C_VEL
LIN {X 0,Y 460.543,Z 293.117,A -85,B 0,C 180,E1 -8128.233,E2 -8128.233} C_VEL
LIN {X 0,Y 460.515,Z 293.117,A -85,B 0,C 180,E1 -8131.283,E2 -8131.283} C_VEL
LIN {X 0,Y 460.526,Z 293.121,A -85,B 0,C 180,E1 -8134.506,E2 -8134.506} C_VEL
LIN {X 0,Y 460.495,Z 293.118,A -85,B 0,C 180,E1 -8137.624,E2 -8137.624} C_VEL
LIN {X 0,Y 460.533,Z 293.115,A -85,B 0,C 180,E1 -8140.269,E2 -8140.269} C_VEL
LIN {X 0,Y 460.493,Z 293.121,A -85,B 0,C 180,E1 -8143.376,E2 -8143.376} C_VEL
LIN {X 0,Y 460.5,Z 293.121,A -85,B 0,C 180,E1 -8146.626,E2 -8146.626} C_VEL
LIN {X 0,Y 460.52,Z 293.116,A -85,B 0,C 180,E1 -8149.734,E2 -8149.734} C_VEL
LIN {X 0,Y 460.495,Z 293.12,A -85,B 0,C 180,E1 -8152.524,E2 -8152.524} C_VEL
LIN {X 0,Y 460.533,Z 293.117,A -85,B 0,C 180,E1 -8155.623,E2 -8155.623} C_VEL
LIN {X 0,Y 460.534,Z 293.115,A -85,B 0,C 180,E1 -8158.745,E2 -8158.745} C_VEL
LIN {X 0,Y 460.506,Z 293.121,A -85,B 0,C 180,E1 -8161.765,E2 -8161.765} C_VEL
LIN {X 0,Y 460.517,Z 293.116,A -85,B 0,C 180,E1 -8164.704,E2 -8164.704} C_VEL
LIN {X 0,Y 460.508,Z 293.126,A -85,B 0,C 180,E1 -8167.572,E2 -8167.572} C_VEL
LIN {X 0,Y 460.565,Z 293.11,A -85,B 0,C 180,E1 -8170.385,E2 -8170.385} C_VEL
LIN {X 0,Y 460.603,Z 293.111,A -85,B 0,C 180,E1 -8174.059,E2 -8174.059} C_VEL
LIN {X 0,Y 460.601,Z 293.114,A -85,B 0,C 180,E1 -8177.666,E2 -8177.666} C_VEL
LIN {X 0,Y 460.588,Z 293.114,A -85,B 0,C 180,E1 -8177.883,E2 -8177.883} C_VEL
LIN {X 0,Y 460.316,Z 293.433,A -85,B 0,C 180,E1 -8178.367,E2 -8178.367} C_VEL
LIN {X 0,Y 459.222,Z 294.886,A -85,B 0,C 180,E1 -8179.066,E2 -8179.066} C_VEL
LIN {X 0,Y 457.716,Z 297.169,A -85,B 0,C 180,E1 -8179.726,E2 -8179.726} C_VEL
LIN {X 0,Y 455.709,Z 301.095,A -85,B 0,C 180,E1 -8180.585,E2 -8180.585} C_VEL
LIN {X 0,Y 454.664,Z 305.401,A -85,B 0,C 180,E1 -8181.441,E2 -8181.441} C_VEL
LIN {X 0,Y 454.455,Z 311.252,A -85,B 0,C 180,E1 -8182.617,E2 -8182.617} C_VEL
LIN {X 0,Y 457.499,Z 327.13,A -85,B 0,C 180,E1 -8182.997,E2 -8182.997} C_VEL
LIN {X 0,Y 456.728,Z 418.589,A -85,B 0,C 180,E1 -8184.454,E2 -8184.454} C_VEL
LIN {X 0,Y 456.437,Z 431.69,A -85,B 0,C 180,E1 -8184.838,E2 -8184.838} C_VEL
LIN {X 0,Y 456.115,Z 444.808,A -85,B 0,C 180,E1 -8185.416,E2 -8185.416} C_VEL
LIN {X 0,Y 455.636,Z 456.675,A -85,B 0,C 180,E1 -8186.131,E2 -8186.131} C_VEL
LIN {X 0,Y 454.999,Z 466.791,A -85,B 0,C 180,E1 -8186.901,E2 -8186.901} C_VEL
LIN {X 0,Y 454.419,Z 477.256,A -85,B 0,C 180,E1 -8187.895,E2 -8187.895} C_VEL
LIN {X 0,Y 454.063,Z 485.797,A -85,B 0,C 180,E1 -8188.892,E2 -8188.892} C_VEL
LIN {X 0,Y 453.669,Z 493.689,A -85,B 0,C 180,E1 -8190,E2 -8190} C_VEL
LIN {X 0,Y 453.249,Z 501.451,A -85,B 0,C 180,E1 -8191.333,E2 -8191.333} C_VEL
LIN {X 0,Y 452.935,Z 507.66,A -85,B 0,C 180,E1 -8192.668,E2 -8192.668} C_VEL
LIN {X 0,Y 452.772,Z 512.602,A -85,B 0,C 180,E1 -8194.006,E2 -8194.006} C_VEL
LIN {X 0,Y 452.663,Z 516.437,A -85,B 0,C 180,E1 -8195.345,E2 -8195.345} C_VEL
LIN {X 0,Y 452.648,Z 518.814,A -85,B 0,C 180,E1 -8196.441,E2 -8196.441} C_VEL
LIN {X 0,Y 452.455,Z 521.133,A -85,B 0,C 180,E1 -8198.036,E2 -8198.036} C_VEL
LIN {X 0,Y 452.383,Z 522.177,A -85,B 0,C 180,E1 -8199.84,E2 -8199.84} C_VEL
LIN {X 0,Y 452.444,Z 522.116,A -85,B 0,C 180,E1 -8200.743,E2 -8200.743} C_VEL
LIN {X 0,Y 452.511,Z 521.396,A -85,B 0,C 180,E1 -8201.914,E2 -8201.914} C_VEL
LIN {X 0,Y 452.482,Z 519.405,A -85,B 0,C 180,E1 -8203.473,E2 -8203.473} C_VEL
LIN {X 0,Y 452.672,Z 516.591,A -85,B 0,C 180,E1 -8204.843,E2 -8204.843} C_VEL
LIN {X 0,Y 452.839,Z 512.701,A -85,B 0,C 180,E1 -8206.222,E2 -8206.222} C_VEL
LIN {X 0,Y 453.088,Z 507.614,A -85,B 0,C 180,E1 -8207.606,E2 -8207.606} C_VEL
LIN {X 0,Y 453.49,Z 500.953,A -85,B 0,C 180,E1 -8209.03,E2 -8209.03} C_VEL
LIN {X 0,Y 453.915,Z 492.955,A -85,B 0,C 180,E1 -8210.388,E2 -8210.388} C_VEL
LIN {X 0,Y 454.457,Z 484.536,A -85,B 0,C 180,E1 -8211.548,E2 -8211.548} C_VEL
LIN {X 0,Y 454.985,Z 475.251,A -85,B 0,C 180,E1 -8212.6,E2 -8212.6} C_VEL
LIN {X 0,Y 455.543,Z 465.178,A -85,B 0,C 180,E1 -8213.528,E2 -8213.528} C_VEL
LIN {X 0,Y 456.113,Z 454.068,A -85,B 0,C 180,E1 -8214.342,E2 -8214.342} C_VEL
LIN {X 0,Y 456.589,Z 441.706,A -85,B 0,C 180,E1 -8215.042,E2 -8215.042} C_VEL
LIN {X 0,Y 456.912,Z 429.699,A -85,B 0,C 180,E1 -8215.541,E2 -8215.541} C_VEL
LIN {X 0,Y 457.135,Z 418.169,A -85,B 0,C 180,E1 -8215.864,E2 -8215.864} C_VEL
LIN {X 0,Y 458.063,Z 327.474,A -85,B 0,C 180,E1 -8217.319,E2 -8217.319} C_VEL
LIN {X 0,Y 454.706,Z 311.295,A -85,B 0,C 180,E1 -8217.75,E2 -8217.75} C_VEL
LIN {X 0,Y 454.9,Z 301.955,A -85,B 0,C 180,E1 -8219.629,E2 -8219.629} C_VEL
LIN {X 0,Y 453.53,Z 294.195,A -85,B 0,C 180,E1 -8221.298,E2 -8221.298} C_VEL
LIN {X 0,Y 453.476,Z 294.001,A -85,B 0,C 180,E1 -8223.913,E2 -8223.913} C_VEL
LIN {X 0,Y 453.451,Z 293.993,A -85,B 0,C 180,E1 -8227.19,E2 -8227.19} C_VEL
LIN {X 0,Y 453.485,Z 293.995,A -85,B 0,C 180,E1 -8229.45,E2 -8229.45} C_VEL
LIN {X 0,Y 453.476,Z 293.996,A -85,B 0,C 180,E1 -8231.935,E2 -8231.935} C_VEL
LIN {X 0,Y 453.483,Z 293.994,A -85,B 0,C 180,E1 -8235.471,E2 -8235.471} C_VEL
LIN {X 0,Y 453.478,Z 293.995,A -85,B 0,C 180,E1 -8238.209,E2 -8238.209} C_VEL
LIN {X 0,Y 453.509,Z 293.995,A -85,B 0,C 180,E1 -8240.791,E2 -8240.791} C_VEL
LIN {X 0,Y 453.453,Z 293.994,A -85,B 0,C 180,E1 -8243.917,E2 -8243.917} C_VEL
LIN {X 0,Y 453.482,Z 293.996,A -85,B 0,C 180,E1 -8247.151,E2 -8247.151} C_VEL
LIN {X 0,Y 453.474,Z 293.99,A -85,B 0,C 180,E1 -8250.268,E2 -8250.268} C_VEL
LIN {X 0,Y 453.503,Z 293.992,A -85,B 0,C 180,E1 -8253.294,E2 -8253.294} C_VEL
LIN {X 0,Y 453.501,Z 293.985,A -85,B 0,C 180,E1 -8256.239,E2 -8256.239} C_VEL
LIN {X 0,Y 453.482,Z 293.996,A -85,B 0,C 180,E1 -8259.118,E2 -8259.118} C_VEL
LIN {X 0,Y 453.51,Z 293.992,A -85,B 0,C 180,E1 -8261.945,E2 -8261.945} C_VEL
LIN {X 0,Y 453.539,Z 293.982,A -85,B 0,C 180,E1 -8264.726,E2 -8264.726} C_VEL
LIN {X 0,Y 453.559,Z 293.981,A -85,B 0,C 180,E1 -8268.379,E2 -8268.379} C_VEL
LIN {X 0,Y 453.651,Z 293.975,A -85,B 0,C 180,E1 -8271.985,E2 -8271.985} C_VEL
LIN {X 0,Y 453.666,Z 293.969,A -85,B 0,C 180,E1 -8274.667,E2 -8274.667} C_VEL
LIN {X 0,Y 453.744,Z 293.96,A -85,B 0,C 180,E1 -8277.337,E2 -8277.337} C_VEL
LIN {X 0,Y 453.822,Z 293.956,A -85,B 0,C 180,E1 -8280,E2 -8280} C_VEL
LIN {X 0,Y 453.743,Z 293.958,A -85,B 0,C 180,E1 -8282.664,E2 -8282.664} C_VEL
LIN {X 0,Y 453.668,Z 293.972,A -85,B 0,C 180,E1 -8286.226,E2 -8286.226} C_VEL
LIN {X 0,Y 453.592,Z 293.979,A -85,B 0,C 180,E1 -8288.914,E2 -8288.914} C_VEL
LIN {X 0,Y 453.563,Z 293.986,A -85,B 0,C 180,E1 -8292.529,E2 -8292.529} C_VEL
LIN {X 0,Y 453.545,Z 293.986,A -85,B 0,C 180,E1 -8296.196,E2 -8296.196} C_VEL
LIN {X 0,Y 453.52,Z 293.989,A -85,B 0,C 180,E1 -8299.041,E2 -8299.041} C_VEL
LIN {X 0,Y 453.477,Z 293.993,A -85,B 0,C 180,E1 -8301.836,E2 -8301.836} C_VEL
LIN {X 0,Y 453.514,Z 293.992,A -85,B 0,C 180,E1 -8304.735,E2 -8304.735} C_VEL
LIN {X 0,Y 453.533,Z 293.985,A -85,B 0,C 180,E1 -8307.96,E2 -8307.96} C_VEL
LIN {X 0,Y 453.466,Z 293.995,A -85,B 0,C 180,E1 -8311.525,E2 -8311.525} C_VEL
LIN {X 0,Y 453.488,Z 293.996,A -85,B 0,C 180,E1 -8314.777,E2 -8314.777} C_VEL
LIN {X 0,Y 453.464,Z 293.994,A -85,B 0,C 180,E1 -8318.312,E2 -8318.312} C_VEL
LIN {X 0,Y 453.495,Z 293.981,A -85,B 0,C 180,E1 -8320.609,E2 -8320.609} C_VEL
LIN {X 0,Y 453.456,Z 294.002,A -85,B 0,C 180,E1 -8323.244,E2 -8323.244} C_VEL
LIN {X 0,Y 453.463,Z 294,A -85,B 0,C 180,E1 -8325.779,E2 -8325.779} C_VEL
LIN {X 0,Y 453.481,Z 293.995,A -85,B 0,C 180,E1 -8328.209,E2 -8328.209} C_VEL
LIN {X 0,Y 453.489,Z 293.993,A -85,B 0,C 180,E1 -8330.795,E2 -8330.795} C_VEL
LIN {X 0,Y 453.456,Z 294.003,A -85,B 0,C 180,E1 -8333.917,E2 -8333.917} C_VEL
LIN {X 0,Y 453.485,Z 293.996,A -85,B 0,C 180,E1 -8337.151,E2 -8337.151} C_VEL
LIN {X 0,Y 453.477,Z 293.999,A -85,B 0,C 180,E1 -8340.268,E2 -8340.268} C_VEL
LIN {X 0,Y 453.579,Z 294.164,A -85,B 0,C 180,E1 -8343.298,E2 -8343.298} C_VEL
LIN {X 0,Y 455.937,Z 305.802,A -85,B 0,C 180,E1 -8345.63,E2 -8345.63} C_VEL
LIN {X 0,Y 456.113,Z 309.808,A -85,B 0,C 180,E1 -8346.383,E2 -8346.383} C_VEL
LIN {X 0,Y 455.136,Z 328.036,A -85,B 0,C 180,E1 -8349.669,E2 -8349.669} C_VEL
LIN {X 0,Y 454.449,Z 342.816,A -85,B 0,C 180,E1 -8352.297,E2 -8352.297} C_VEL
LIN {X 0,Y 457.79,Z 363.659,A -85,B 0,C 180,E1 -8352.787,E2 -8352.787} C_VEL
LIN {X 0,Y 457.076,Z 451.942,A -85,B 0,C 180,E1 -8354.219,E2 -8354.219} C_VEL
LIN {X 0,Y 456.632,Z 464.198,A -85,B 0,C 180,E1 -8354.575,E2 -8354.575} C_VEL
LIN {X 0,Y 456.114,Z 477.54,A -85,B 0,C 180,E1 -8355.157,E2 -8355.157} C_VEL
LIN {X 0,Y 455.565,Z 488.758,A -85,B 0,C 180,E1 -8355.824,E2 -8355.824} C_VEL
LIN {X 0,Y 454.951,Z 500.316,A -85,B 0,C 180,E1 -8356.71,E2 -8356.71} C_VEL
LIN {X 0,Y 454.391,Z 510.853,A -85,B 0,C 180,E1 -8357.721,E2 -8357.721} C_VEL
LIN {X 0,Y 453.815,Z 520.304,A -85,B 0,C 180,E1 -8358.838,E2 -8358.838} C_VEL
LIN {X 0,Y 453.303,Z 529.421,A -85,B 0,C 180,E1 -8360.18,E2 -8360.18} C_VEL
LIN {X 0,Y 452.95,Z 536.784,A -85,B 0,C 180,E1 -8361.523,E2 -8361.523} C_VEL
LIN {X 0,Y 452.716,Z 542.701,A -85,B 0,C 180,E1 -8362.866,E2 -8362.866} C_VEL
LIN {X 0,Y 452.557,Z 547.376,A -85,B 0,C 180,E1 -8364.206,E2 -8364.206} C_VEL
LIN {X 0,Y 452.487,Z 550.946,A -85,B 0,C 180,E1 -8365.546,E2 -8365.546} C_VEL
LIN {X 0,Y 452.482,Z 552.777,A -85,B 0,C 180,E1 -8366.438,E2 -8366.438} C_VEL
LIN {X 0,Y 452.508,Z 554.155,A -85,B 0,C 180,E1 -8367.329,E2 -8367.329} C_VEL
LIN {X 0,Y 452.43,Z 555.73,A -85,B 0,C 180,E1 -8369.11,E2 -8369.11} C_VEL
LIN {X 0,Y 452.465,Z 555.92,A -85,B 0,C 180,E1 -8370,E2 -8370} C_VEL
LIN {X 0,Y 452.457,Z 555.056,A -85,B 0,C 180,E1 -8371.78,E2 -8371.78} C_VEL
LIN {X 0,Y 452.508,Z 554.042,A -85,B 0,C 180,E1 -8372.67,E2 -8372.67} C_VEL
LIN {X 0,Y 452.484,Z 552.607,A -85,B 0,C 180,E1 -8373.562,E2 -8373.562} C_VEL
LIN {X 0,Y 452.545,Z 549.626,A -85,B 0,C 180,E1 -8374.9,E2 -8374.9} C_VEL
LIN {X 0,Y 452.611,Z 545.027,A -85,B 0,C 180,E1 -8376.396,E2 -8376.396} C_VEL
LIN {X 0,Y 452.841,Z 538.352,A -85,B 0,C 180,E1 -8378.029,E2 -8378.029} C_VEL
LIN {X 0,Y 453.128,Z 531.335,A -85,B 0,C 180,E1 -8379.372,E2 -8379.372} C_VEL
LIN {X 0,Y 453.55,Z 522.534,A -85,B 0,C 180,E1 -8380.716,E2 -8380.716} C_VEL
LIN {X 0,Y 454.141,Z 512.539,A -85,B 0,C 180,E1 -8381.945,E2 -8381.945} C_VEL
LIN {X 0,Y 454.606,Z 502.436,A -85,B 0,C 180,E1 -8382.946,E2 -8382.946} C_VEL
LIN {X 0,Y 455.165,Z 491.031,A -85,B 0,C 180,E1 -8383.846,E2 -8383.846} C_VEL
LIN {X 0,Y 455.707,Z 479.303,A -85,B 0,C 180,E1 -8384.57,E2 -8384.57} C_VEL
LIN {X 0,Y 456.192,Z 466.566,A -85,B 0,C 180,E1 -8385.154,E2 -8385.154} C_VEL
LIN {X 0,Y 456.592,Z 454.144,A -85,B 0,C 180,E1 -8385.54,E2 -8385.54} C_VEL
LIN {X 0,Y 456.855,Z 433.65,A -85,B 0,C 180,E1 -8385.903,E2 -8385.903} C_VEL
LIN {X 0,Y 457.311,Z 363.451,A -85,B 0,C 180,E1 -8387.008,E2 -8387.008} C_VEL
LIN {X 0,Y 454.254,Z 343.068,A -85,B 0,C 180,E1 -8387.441,E2 -8387.441} C_VEL
LIN {X 0,Y 455.107,Z 323.917,A -85,B 0,C 180,E1 -8390.804,E2 -8390.804} C_VEL
LIN {X 0,Y 455.873,Z 306.81,A -85,B 0,C 180,E1 -8393.846,E2 -8393.846} C_VEL
LIN {X 0,Y 453.928,Z 295.932,A -85,B 0,C 180,E1 -8395.919,E2 -8395.919} C_VEL
LIN {X 0,Y 453.54,Z 293.991,A -85,B 0,C 180,E1 -8396.322,E2 -8396.322} C_VEL
LIN {X 0,Y 453.51,Z 293.994,A -85,B 0,C 180,E1 -8398.711,E2 -8398.711} C_VEL
LIN {X 0,Y 453.464,Z 293.998,A -85,B 0,C 180,E1 -8401.799,E2 -8401.799} C_VEL
LIN {X 0,Y 453.479,Z 293.993,A -85,B 0,C 180,E1 -8404.989,E2 -8404.989} C_VEL
LIN {X 0,Y 453.459,Z 294.004,A -85,B 0,C 180,E1 -8408.311,E2 -8408.311} C_VEL
LIN {X 0,Y 453.492,Z 293.996,A -85,B 0,C 180,E1 -8410.608,E2 -8410.608} C_VEL
LIN {X 0,Y 453.452,Z 293.996,A -85,B 0,C 180,E1 -8413.243,E2 -8413.243} C_VEL
LIN {X 0,Y 453.461,Z 293.995,A -85,B 0,C 180,E1 -8415.778,E2 -8415.778} C_VEL
LIN {X 0,Y 453.477,Z 293.996,A -85,B 0,C 180,E1 -8418.209,E2 -8418.209} C_VEL
LIN {X 0,Y 453.507,Z 293.996,A -85,B 0,C 180,E1 -8420.79,E2 -8420.79} C_VEL
LIN {X 0,Y 453.451,Z 293.996,A -85,B 0,C 180,E1 -8423.917,E2 -8423.917} C_VEL
LIN {X 0,Y 453.479,Z 293.997,A -85,B 0,C 180,E1 -8427.151,E2 -8427.151} C_VEL
LIN {X 0,Y 453.471,Z 293.994,A -85,B 0,C 180,E1 -8430.268,E2 -8430.268} C_VEL
LIN {X 0,Y 453.503,Z 293.994,A -85,B 0,C 180,E1 -8433.293,E2 -8433.293} C_VEL
LIN {X 0,Y 453.499,Z 293.99,A -85,B 0,C 180,E1 -8436.238,E2 -8436.238} C_VEL
LIN {X 0,Y 453.479,Z 294.001,A -85,B 0,C 180,E1 -8439.117,E2 -8439.117} C_VEL
LIN {X 0,Y 453.507,Z 293.99,A -85,B 0,C 180,E1 -8441.944,E2 -8441.944} C_VEL
LIN {X 0,Y 453.537,Z 293.987,A -85,B 0,C 180,E1 -8444.726,E2 -8444.726} C_VEL
LIN {X 0,Y 453.555,Z 293.983,A -85,B 0,C 180,E1 -8448.379,E2 -8448.379} C_VEL
LIN {X 0,Y 453.647,Z 293.974,A -85,B 0,C 180,E1 -8451.985,E2 -8451.985} C_VEL
LIN {X 0,Y 453.664,Z 293.969,A -85,B 0,C 180,E1 -8454.666,E2 -8454.666} C_VEL
LIN {X 0,Y 453.738,Z 293.964,A -85,B 0,C 180,E1 -8457.336,E2 -8457.336} C_VEL
LIN {X 0,Y 453.816,Z 293.955,A -85,B 0,C 180,E1 -8460,E2 -8460} C_VEL
LIN {X 0,Y 453.739,Z 293.96,A -85,B 0,C 180,E1 -8462.663,E2 -8462.663} C_VEL
LIN {X 0,Y 453.646,Z 293.976,A -85,B 0,C 180,E1 -8466.226,E2 -8466.226} C_VEL
LIN {X 0,Y 453.586,Z 293.979,A -85,B 0,C 180,E1 -8468.913,E2 -8468.913} C_VEL
LIN {X 0,Y 453.558,Z 293.985,A -85,B 0,C 180,E1 -8472.529,E2 -8472.529} C_VEL
LIN {X 0,Y 453.539,Z 293.994,A -85,B 0,C 180,E1 -8476.196,E2 -8476.196} C_VEL
LIN {X 0,Y 453.511,Z 293.989,A -85,B 0,C 180,E1 -8479.039,E2 -8479.039} C_VEL
LIN {X 0,Y 453.471,Z 293.996,A -85,B 0,C 180,E1 -8481.836,E2 -8481.836} C_VEL
LIN {X 0,Y 453.494,Z 293.995,A -85,B 0,C 180,E1 -8484.735,E2 -8484.735} C_VEL
LIN {X 0,Y 453.523,Z 293.989,A -85,B 0,C 180,E1 -8487.959,E2 -8487.959} C_VEL
LIN {X 0,Y 453.46,Z 293.995,A -85,B 0,C 180,E1 -8491.525,E2 -8491.525} C_VEL
LIN {X 0,Y 453.482,Z 293.999,A -85,B 0,C 180,E1 -8494.778,E2 -8494.778} C_VEL
LIN {X 0,Y 453.457,Z 293.998,A -85,B 0,C 180,E1 -8498.312,E2 -8498.312} C_VEL
LIN {X 0,Y 453.489,Z 293.997,A -85,B 0,C 180,E1 -8500.609,E2 -8500.609} C_VEL
LIN {X 0,Y 453.45,Z 294,A -85,B 0,C 180,E1 -8503.244,E2 -8503.244} C_VEL
LIN {X 0,Y 453.457,Z 293.995,A -85,B 0,C 180,E1 -8505.779,E2 -8505.779} C_VEL
LIN {X 0,Y 453.466,Z 293.998,A -85,B 0,C 180,E1 -8509.413,E2 -8509.413} C_VEL
LIN {X 0,Y 453.448,Z 294,A -85,B 0,C 180,E1 -8512.811,E2 -8512.811} C_VEL
LIN {X 0,Y 453.465,Z 293.994,A -85,B 0,C 180,E1 -8516.087,E2 -8516.087} C_VEL
LIN {X 0,Y 453.471,Z 294.001,A -85,B 0,C 180,E1 -8519.241,E2 -8519.241} C_VEL
LIN {X 0,Y 453.472,Z 293.993,A -85,B 0,C 180,E1 -8522.294,E2 -8522.294} C_VEL
LIN {X 0,Y 453.465,Z 293.999,A -85,B 0,C 180,E1 -8525.263,E2 -8525.263} C_VEL
LIN {X 0,Y 453.479,Z 293.993,A -85,B 0,C 180,E1 -8528.416,E2 -8528.416} C_VEL
LIN {X 0,Y 453.521,Z 293.988,A -85,B 0,C 180,E1 -8531.009,E2 -8531.009} C_VEL
LIN {X 0,Y 453.568,Z 293.989,A -85,B 0,C 180,E1 -8533.88,E2 -8533.88} C_VEL
LIN {X 0,Y 453.563,Z 293.988,A -85,B 0,C 180,E1 -8537.472,E2 -8537.472} C_VEL
LIN {X 0,Y 453.551,Z 294.044,A -85,B 0,C 180,E1 -8539.058,E2 -8539.058} C_VEL
LIN {X 0,Y 454.657,Z 301.577,A -85,B 0,C 180,E1 -8540.66,E2 -8540.66} C_VEL
LIN {X 0,Y 454.664,Z 305.401,A -85,B 0,C 180,E1 -8541.441,E2 -8541.441} C_VEL
LIN {X 0,Y 454.408,Z 307.858,A -85,B 0,C 180,E1 -8541.814,E2 -8541.814} C_VEL
LIN {X 0,Y 453.924,Z 310.902,A -85,B 0,C 180,E1 -8542.111,E2 -8542.111} C_VEL
LIN {X 0,Y 452.967,Z 316.141,A -85,B 0,C 180,E1 -8542.432,E2 -8542.432} C_VEL
LIN {X 0,Y 451.933,Z 321.942,A -85,B 0,C 180,E1 -8542.638,E2 -8542.638} C_VEL
LIN {X 0,Y 451.326,Z 325.974,A -85,B 0,C 180,E1 -8542.733,E2 -8542.733} C_VEL
LIN {X 0,Y 450.703,Z 334.167,A -85,B 0,C 180,E1 -8542.872,E2 -8542.872} C_VEL
LIN {X 0,Y 449.839,Z 419.525,A -85,B 0,C 180,E1 -8544.256,E2 -8544.256} C_VEL
LIN {X 0,Y 449.518,Z 433.158,A -85,B 0,C 180,E1 -8544.674,E2 -8544.674} C_VEL
LIN {X 0,Y 449.2,Z 445.399,A -85,B 0,C 180,E1 -8545.233,E2 -8545.233} C_VEL
LIN {X 0,Y 448.703,Z 457.18,A -85,B 0,C 180,E1 -8545.959,E2 -8545.959} C_VEL
LIN {X 0,Y 448.03,Z 467.259,A -85,B 0,C 180,E1 -8546.741,E2 -8546.741} C_VEL
LIN {X 0,Y 447.438,Z 477.691,A -85,B 0,C 180,E1 -8547.75,E2 -8547.75} C_VEL
LIN {X 0,Y 447.022,Z 487.085,A -85,B 0,C 180,E1 -8548.874,E2 -8548.874} C_VEL
LIN {X 0,Y 446.54,Z 496.153,A -85,B 0,C 180,E1 -8550.226,E2 -8550.226} C_VEL
LIN {X 0,Y 446.085,Z 503.477,A -85,B 0,C 180,E1 -8551.58,E2 -8551.58} C_VEL
LIN {X 0,Y 445.828,Z 510.208,A -85,B 0,C 180,E1 -8553.163,E2 -8553.163} C_VEL
LIN {X 0,Y 445.561,Z 514.669,A -85,B 0,C 180,E1 -8554.524,E2 -8554.524} C_VEL
LIN {X 0,Y 445.593,Z 517.013,A -85,B 0,C 180,E1 -8555.43,E2 -8555.43} C_VEL
LIN {X 0,Y 445.576,Z 519.14,A -85,B 0,C 180,E1 -8556.441,E2 -8556.441} C_VEL
LIN {X 0,Y 445.35,Z 521.517,A -85,B 0,C 180,E1 -8558.165,E2 -8558.165} C_VEL
LIN {X 0,Y 445.308,Z 522.466,A -85,B 0,C 180,E1 -8559.998,E2 -8559.998} C_VEL
LIN {X 0,Y 445.356,Z 522.341,A -85,B 0,C 180,E1 -8560.916,E2 -8560.916} C_VEL
LIN {X 0,Y 445.427,Z 521.657,A -85,B 0,C 180,E1 -8561.974,E2 -8561.974} C_VEL
LIN {X 0,Y 445.43,Z 519.454,A -85,B 0,C 180,E1 -8563.69,E2 -8563.69} C_VEL
LIN {X 0,Y 445.635,Z 516.538,A -85,B 0,C 180,E1 -8565.083,E2 -8565.083} C_VEL
LIN {X 0,Y 445.806,Z 512.54,A -85,B 0,C 180,E1 -8566.485,E2 -8566.485} C_VEL
LIN {X 0,Y 446.166,Z 506.297,A -85,B 0,C 180,E1 -8568.126,E2 -8568.126} C_VEL
LIN {X 0,Y 446.613,Z 499.414,A -85,B 0,C 180,E1 -8569.536,E2 -8569.536} C_VEL
LIN {X 0,Y 446.998,Z 492.329,A -85,B 0,C 180,E1 -8570.718,E2 -8570.718} C_VEL
LIN {X 0,Y 447.59,Z 483.734,A -85,B 0,C 180,E1 -8571.896,E2 -8571.896} C_VEL
LIN {X 0,Y 448.172,Z 474.214,A -85,B 0,C 180,E1 -8572.959,E2 -8572.959} C_VEL
LIN {X 0,Y 448.809,Z 463.753,A -85,B 0,C 180,E1 -8573.903,E2 -8573.903} C_VEL
LIN {X 0,Y 449.362,Z 452.735,A -85,B 0,C 180,E1 -8574.698,E2 -8574.698} C_VEL
LIN {X 0,Y 449.863,Z 440.437,A -85,B 0,C 180,E1 -8575.382,E2 -8575.382} C_VEL
LIN {X 0,Y 450.189,Z 427.591,A -85,B 0,C 180,E1 -8575.889,E2 -8575.889} C_VEL
LIN {X 0,Y 450.45,Z 416.053,A -85,B 0,C 180,E1 -8576.184,E2 -8576.184} C_VEL
LIN {X 0,Y 451.404,Z 328.618,A -85,B 0,C 180,E1 -8577.6,E2 -8577.6} C_VEL
LIN {X 0,Y 447.825,Z 311.58,A -85,B 0,C 180,E1 -8578.06,E2 -8578.06} C_VEL
LIN {X 0,Y 447.939,Z 302.699,A -85,B 0,C 180,E1 -8579.877,E2 -8579.877} C_VEL
LIN {X 0,Y 446.458,Z 294.874,A -85,B 0,C 180,E1 -8581.605,E2 -8581.605} C_VEL
LIN {X 0,Y 446.429,Z 294.88,A -85,B 0,C 180,E1 -8584.523,E2 -8584.523} C_VEL
LIN {X 0,Y 446.414,Z 294.872,A -85,B 0,C 180,E1 -8588.079,E2 -8588.079} C_VEL
LIN {X 0,Y 446.426,Z 294.877,A -85,B 0,C 180,E1 -8590.918,E2 -8590.918} C_VEL
LIN {X 0,Y 446.399,Z 294.877,A -85,B 0,C 180,E1 -8593.846,E2 -8593.846} C_VEL
LIN {X 0,Y 446.398,Z 294.881,A -85,B 0,C 180,E1 -8596.403,E2 -8596.403} C_VEL
LIN {X 0,Y 446.426,Z 294.876,A -85,B 0,C 180,E1 -8599.082,E2 -8599.082} C_VEL
LIN {X 0,Y 446.414,Z 294.871,A -85,B 0,C 180,E1 -8601.921,E2 -8601.921} C_VEL
LIN {X 0,Y 446.428,Z 294.871,A -85,B 0,C 180,E1 -8605.477,E2 -8605.477} C_VEL
LIN {X 0,Y 446.415,Z 294.873,A -85,B 0,C 180,E1 -8608.7,E2 -8608.7} C_VEL
LIN {X 0,Y 446.484,Z 294.86,A -85,B 0,C 180,E1 -8611.821,E2 -8611.821} C_VEL
LIN {X 0,Y 446.449,Z 294.869,A -85,B 0,C 180,E1 -8614.847,E2 -8614.847} C_VEL
LIN {X 0,Y 446.447,Z 294.868,A -85,B 0,C 180,E1 -8618.245,E2 -8618.245} C_VEL
LIN {X 0,Y 446.456,Z 294.874,A -85,B 0,C 180,E1 -8621.649,E2 -8621.649} C_VEL
LIN {X 0,Y 446.507,Z 294.858,A -85,B 0,C 180,E1 -8624.48,E2 -8624.48} C_VEL
LIN {X 0,Y 446.517,Z 294.859,A -85,B 0,C 180,E1 -8628.193,E2 -8628.193} C_VEL
LIN {X 0,Y 446.6,Z 294.855,A -85,B 0,C 180,E1 -8631.858,E2 -8631.858} C_VEL
LIN {X 0,Y 446.64,Z 294.845,A -85,B 0,C 180,E1 -8634.583,E2 -8634.583} C_VEL
LIN {X 0,Y 446.664,Z 294.844,A -85,B 0,C 180,E1 -8638.197,E2 -8638.197} C_VEL
LIN {X 0,Y 446.792,Z 294.832,A -85,B 0,C 180,E1 -8640,E2 -8640} C_VEL
LIN {X 0,Y 446.69,Z 294.836,A -85,B 0,C 180,E1 -8642.706,E2 -8642.706} C_VEL
LIN {X 0,Y 446.638,Z 294.846,A -85,B 0,C 180,E1 -8646.324,E2 -8646.324} C_VEL
LIN {X 0,Y 446.537,Z 294.857,A -85,B 0,C 180,E1 -8649.056,E2 -8649.056} C_VEL
LIN {X 0,Y 446.521,Z 294.863,A -85,B 0,C 180,E1 -8652.73,E2 -8652.73} C_VEL
LIN {X 0,Y 446.496,Z 294.864,A -85,B 0,C 180,E1 -8656.228,E2 -8656.228} C_VEL
LIN {X 0,Y 446.469,Z 294.865,A -85,B 0,C 180,E1 -8659.303,E2 -8659.303} C_VEL
LIN {X 0,Y 446.418,Z 294.874,A -85,B 0,C 180,E1 -8662.2,E2 -8662.2} C_VEL
LIN {X 0,Y 446.458,Z 294.871,A -85,B 0,C 180,E1 -8665.153,E2 -8665.153} C_VEL
LIN {X 0,Y 446.485,Z 294.864,A -85,B 0,C 180,E1 -8668.179,E2 -8668.179} C_VEL
LIN {X 0,Y 446.419,Z 294.871,A -85,B 0,C 180,E1 -8671.775,E2 -8671.775} C_VEL
LIN {X 0,Y 446.429,Z 294.873,A -85,B 0,C 180,E1 -8674.523,E2 -8674.523} C_VEL
LIN {X 0,Y 446.415,Z 294.873,A -85,B 0,C 180,E1 -8678.079,E2 -8678.079} C_VEL
LIN {X 0,Y 446.428,Z 294.863,A -85,B 0,C 180,E1 -8680.918,E2 -8680.918} C_VEL
LIN {X 0,Y 446.401,Z 294.876,A -85,B 0,C 180,E1 -8683.846,E2 -8683.846} C_VEL
LIN {X 0,Y 446.397,Z 294.876,A -85,B 0,C 180,E1 -8686.404,E2 -8686.404} C_VEL
LIN {X 0,Y 446.428,Z 294.875,A -85,B 0,C 180,E1 -8689.083,E2 -8689.083} C_VEL
LIN {X 0,Y 446.409,Z 294.874,A -85,B 0,C 180,E1 -8692.121,E2 -8692.121} C_VEL
LIN {X 0,Y 446.431,Z 294.875,A -85,B 0,C 180,E1 -8695.477,E2 -8695.477} C_VEL
LIN {X 0,Y 446.418,Z 294.876,A -85,B 0,C 180,E1 -8698.7,E2 -8698.7} C_VEL
LIN {X 0,Y 446.487,Z 294.87,A -85,B 0,C 180,E1 -8701.821,E2 -8701.821} C_VEL
LIN {X 0,Y 446.523,Z 294.992,A -85,B 0,C 180,E1 -8703.011,E2 -8703.011} C_VEL
LIN {X 0,Y 448.808,Z 305.989,A -85,B 0,C 180,E1 -8705.263,E2 -8705.263} C_VEL
LIN {X 0,Y 449.228,Z 311.049,A -85,B 0,C 180,E1 -8706.243,E2 -8706.243} C_VEL
LIN {X 0,Y 448.276,Z 327.961,A -85,B 0,C 180,E1 -8709.344,E2 -8709.344} C_VEL
LIN {X 0,Y 447.527,Z 342.542,A -85,B 0,C 180,E1 -8711.981,E2 -8711.981} C_VEL
LIN {X 0,Y 451.078,Z 364.464,A -85,B 0,C 180,E1 -8712.509,E2 -8712.509} C_VEL
LIN {X 0,Y 450.323,Z 451.72,A -85,B 0,C 180,E1 -8713.947,E2 -8713.947} C_VEL
LIN {X 0,Y 449.851,Z 463.956,A -85,B 0,C 180,E1 -8714.307,E2 -8714.307} C_VEL
LIN {X 0,Y 449.3,Z 476.724,A -85,B 0,C 180,E1 -8714.869,E2 -8714.869} C_VEL
LIN {X 0,Y 448.673,Z 488.89,A -85,B 0,C 180,E1 -8715.601,E2 -8715.601} C_VEL
LIN {X 0,Y 448.029,Z 500.62,A -85,B 0,C 180,E1 -8716.523,E2 -8716.523} C_VEL
LIN {X 0,Y 447.442,Z 510.844,A -85,B 0,C 180,E1 -8717.527,E2 -8717.527} C_VEL
LIN {X 0,Y 446.842,Z 520.234,A -85,B 0,C 180,E1 -8718.661,E2 -8718.661} C_VEL
LIN {X 0,Y 446.286,Z 529.31,A -85,B 0,C 180,E1 -8720.024,E2 -8720.024} C_VEL
LIN {X 0,Y 445.885,Z 536.642,A -85,B 0,C 180,E1 -8721.388,E2 -8721.388} C_VEL
LIN {X 0,Y 445.633,Z 542.533,A -85,B 0,C 180,E1 -8722.752,E2 -8722.752} C_VEL
LIN {X 0,Y 445.47,Z 546.686,A -85,B 0,C 180,E1 -8723.955,E2 -8723.955} C_VEL
LIN {X 0,Y 445.412,Z 550.737,A -85,B 0,C 180,E1 -8725.475,E2 -8725.475} C_VEL
LIN {X 0,Y 445.38,Z 552.549,A -85,B 0,C 180,E1 -8726.381,E2 -8726.381} C_VEL
LIN {X 0,Y 445.433,Z 553.919,A -85,B 0,C 180,E1 -8727.287,E2 -8727.287} C_VEL
LIN {X 0,Y 445.341,Z 555.478,A -85,B 0,C 180,E1 -8729.095,E2 -8729.095} C_VEL
LIN {X 0,Y 445.371,Z 555.651,A -85,B 0,C 180,E1 -8730,E2 -8730} C_VEL
LIN {X 0,Y 445.374,Z 554.771,A -85,B 0,C 180,E1 -8731.808,E2 -8731.808} C_VEL
LIN {X 0,Y 445.433,Z 553.75,A -85,B 0,C 180,E1 -8732.713,E2 -8732.713} C_VEL
LIN {X 0,Y 445.384,Z 552.296,A -85,B 0,C 180,E1 -8733.618,E2 -8733.618} C_VEL
LIN {X 0,Y 445.474,Z 549.3,A -85,B 0,C 180,E1 -8734.977,E2 -8734.977} C_VEL
LIN {X 0,Y 445.557,Z 543.777,A -85,B 0,C 180,E1 -8736.748,E2 -8736.748} C_VEL
LIN {X 0,Y 445.768,Z 537.976,A -85,B 0,C 180,E1 -8738.157,E2 -8738.157} C_VEL
LIN {X 0,Y 446.071,Z 530.921,A -85,B 0,C 180,E1 -8739.522,E2 -8739.522} C_VEL
LIN {X 0,Y 446.544,Z 522.081,A -85,B 0,C 180,E1 -8740.886,E2 -8740.886} C_VEL
LIN {X 0,Y 447.142,Z 512.041,A -85,B 0,C 180,E1 -8742.135,E2 -8742.135} C_VEL
LIN {X 0,Y 447.621,Z 501.859,A -85,B 0,C 180,E1 -8743.151,E2 -8743.151} C_VEL
LIN {X 0,Y 448.212,Z 490.379,A -85,B 0,C 180,E1 -8744.066,E2 -8744.066} C_VEL
LIN {X 0,Y 448.793,Z 478.548,A -85,B 0,C 180,E1 -8744.8,E2 -8744.8} C_VEL
LIN {X 0,Y 449.351,Z 465.549,A -85,B 0,C 180,E1 -8745.39,E2 -8745.39} C_VEL
LIN {X 0,Y 449.732,Z 452.739,A -85,B 0,C 180,E1 -8745.783,E2 -8745.783} C_VEL
LIN {X 0,Y 450.1,Z 418.569,A -85,B 0,C 180,E1 -8746.359,E2 -8746.359} C_VEL
LIN {X 0,Y 450.446,Z 364.085,A -85,B 0,C 180,E1 -8747.231,E2 -8747.231} C_VEL
LIN {X 0,Y 447.254,Z 342.784,A -85,B 0,C 180,E1 -8747.693,E2 -8747.693} C_VEL
LIN {X 0,Y 448.101,Z 324.781,A -85,B 0,C 180,E1 -8750.904,E2 -8750.904} C_VEL
LIN {X 0,Y 448.88,Z 308.86,A -85,B 0,C 180,E1 -8753.775,E2 -8753.775} C_VEL
LIN {X 0,Y 448.227,Z 303.619,A -85,B 0,C 180,E1 -8754.77,E2 -8754.77} C_VEL
LIN {X 0,Y 446.524,Z 294.863,A -85,B 0,C 180,E1 -8756.512,E2 -8756.512} C_VEL
LIN {X 0,Y 446.449,Z 294.873,A -85,B 0,C 180,E1 -8759.209,E2 -8759.209} C_VEL
LIN {X 0,Y 446.422,Z 294.877,A -85,B 0,C 180,E1 -8762.361,E2 -8762.361} C_VEL
LIN {X 0,Y 446.418,Z 294.873,A -85,B 0,C 180,E1 -8765.625,E2 -8765.625} C_VEL
LIN {X 0,Y 446.436,Z 294.871,A -85,B 0,C 180,E1 -8769.027,E2 -8769.027} C_VEL
LIN {X 0,Y 446.432,Z 294.877,A -85,B 0,C 180,E1 -8772.277,E2 -8772.277} C_VEL
LIN {X 0,Y 446.449,Z 294.87,A -85,B 0,C 180,E1 -8775.103,E2 -8775.103} C_VEL
LIN {X 0,Y 446.426,Z 294.88,A -85,B 0,C 180,E1 -8778.608,E2 -8778.608} C_VEL
LIN {X 0,Y 446.452,Z 294.872,A -85,B 0,C 180,E1 -8780.974,E2 -8780.974} C_VEL
LIN {X 0,Y 446.416,Z 294.876,A -85,B 0,C 180,E1 -8784.373,E2 -8784.373} C_VEL
LIN {X 0,Y 446.418,Z 294.872,A -85,B 0,C 180,E1 -8787.638,E2 -8787.638} C_VEL
LIN {X 0,Y 446.445,Z 294.875,A -85,B 0,C 180,E1 -8790.79,E2 -8790.79} C_VEL
LIN {X 0,Y 446.474,Z 294.865,A -85,B 0,C 180,E1 -8793.848,E2 -8793.848} C_VEL
LIN {X 0,Y 446.425,Z 294.876,A -85,B 0,C 180,E1 -8796.823,E2 -8796.823} C_VEL
LIN {X 0,Y 446.44,Z 294.871,A -85,B 0,C 180,E1 -8799.737,E2 -8799.737} C_VEL
LIN {X 0,Y 446.459,Z 294.868,A -85,B 0,C 180,E1 -8802.597,E2 -8802.597} C_VEL
LIN {X 0,Y 446.467,Z 294.873,A -85,B 0,C 180,E1 -8805.412,E2 -8805.412} C_VEL
LIN {X 0,Y 446.513,Z 294.861,A -85,B 0,C 180,E1 -8808.193,E2 -8808.193} C_VEL
LIN {X 0,Y 446.595,Z 294.854,A -85,B 0,C 180,E1 -8811.858,E2 -8811.858} C_VEL
LIN {X 0,Y 446.638,Z 294.845,A -85,B 0,C 180,E1 -8814.582,E2 -8814.582} C_VEL
LIN {X 0,Y 446.658,Z 294.844,A -85,B 0,C 180,E1 -8818.196,E2 -8818.196} C_VEL
LIN {X 0,Y 446.786,Z 294.831,A -85,B 0,C 180,E1 -8820,E2 -8820} C_VEL
LIN {X 0,Y 446.686,Z 294.839,A -85,B 0,C 180,E1 -8822.705,E2 -8822.705} C_VEL
LIN {X 0,Y 446.614,Z 294.851,A -85,B 0,C 180,E1 -8826.324,E2 -8826.324} C_VEL
LIN {X 0,Y 446.532,Z 294.858,A -85,B 0,C 180,E1 -8829.055,E2 -8829.055} C_VEL
LIN {X 0,Y 446.516,Z 294.861,A -85,B 0,C 180,E1 -8832.73,E2 -8832.73} C_VEL
LIN {X 0,Y 446.49,Z 294.871,A -85,B 0,C 180,E1 -8836.227,E2 -8836.227} C_VEL
LIN {X 0,Y 446.462,Z 294.866,A -85,B 0,C 180,E1 -8839.303,E2 -8839.303} C_VEL
LIN {X 0,Y 446.413,Z 294.879,A -85,B 0,C 180,E1 -8842.2,E2 -8842.2} C_VEL
LIN {X 0,Y 446.436,Z 294.87,A -85,B 0,C 180,E1 -8845.153,E2 -8845.153} C_VEL
LIN {X 0,Y 446.479,Z 294.869,A -85,B 0,C 180,E1 -8848.179,E2 -8848.179} C_VEL
LIN {X 0,Y 446.413,Z 294.873,A -85,B 0,C 180,E1 -8851.775,E2 -8851.775} C_VEL
LIN {X 0,Y 446.424,Z 294.878,A -85,B 0,C 180,E1 -8854.523,E2 -8854.523} C_VEL
LIN {X 0,Y 446.409,Z 294.874,A -85,B 0,C 180,E1 -8858.079,E2 -8858.079} C_VEL
LIN {X 0,Y 446.422,Z 294.879,A -85,B 0,C 180,E1 -8860.918,E2 -8860.918} C_VEL
LIN {X 0,Y 446.396,Z 294.875,A -85,B 0,C 180,E1 -8863.846,E2 -8863.846} C_VEL
LIN {X 0,Y 446.389,Z 294.877,A -85,B 0,C 180,E1 -8866.405,E2 -8866.405} C_VEL
LIN {X 0,Y 446.398,Z 294.875,A -85,B 0,C 180,E1 -8869.798,E2 -8869.798} C_VEL
LIN {X 0,Y 446.402,Z 294.874,A -85,B 0,C 180,E1 -8872.121,E2 -8872.121} C_VEL
LIN {X 0,Y 446.419,Z 294.877,A -85,B 0,C 180,E1 -8875.477,E2 -8875.477} C_VEL
LIN {X 0,Y 446.411,Z 294.874,A -85,B 0,C 180,E1 -8878.7,E2 -8878.7} C_VEL
LIN {X 0,Y 446.421,Z 294.875,A -85,B 0,C 180,E1 -8881.837,E2 -8881.837} C_VEL
LIN {X 0,Y 446.417,Z 294.873,A -85,B 0,C 180,E1 -8884.846,E2 -8884.846} C_VEL
LIN {X 0,Y 446.446,Z 294.87,A -85,B 0,C 180,E1 -8888.246,E2 -8888.246} C_VEL
LIN {X 0,Y 446.447,Z 294.877,A -85,B 0,C 180,E1 -8891.649,E2 -8891.649} C_VEL
LIN {X 0,Y 446.506,Z 294.863,A -85,B 0,C 180,E1 -8894.48,E2 -8894.48} C_VEL
LIN {X 0,Y 446.505,Z 294.869,A -85,B 0,C 180,E1 -8898.193,E2 -8898.193} C_VEL
LIN {X 0,Y 446.537,Z 294.981,A -85,B 0,C 180,E1 -8898.913,E2 -8898.913} C_VEL
LIN {X 0,Y 447.683,Z 302.414,A -85,B 0,C 180,E1 -8900.513,E2 -8900.513} C_VEL
LIN {X 0,Y 447.483,Z 311.532,A -85,B 0,C 180,E1 -8902.379,E2 -8902.379} C_VEL
LIN {X 0,Y 450.707,Z 328.385,A -85,B 0,C 180,E1 -8902.778,E2 -8902.778} C_VEL
LIN {X 0,Y 450.703,Z 334.167,A -85,B 0,C 180,E1 -8902.872,E2 -8902.872} C_VEL
LIN {X 0,Y 450.021,Z 340.008,A -85,B 0,C 180,E1 -8902.943,E2 -8902.943} C_VEL
LIN {X 0,Y 444.309,Z 358.989,A -85,B 0,C 180,E1 -8903.054,E2 -8903.054} C_VEL
LIN {X 0,Y 443.596,Z 364.832,A -85,B 0,C 180,E1 -8903.125,E2 -8903.125} C_VEL
LIN {X 0,Y 442.979,Z 419.241,A -85,B 0,C 180,E1 -8904.024,E2 -8904.024} C_VEL
LIN {X 0,Y 442.664,Z 432.307,A -85,B 0,C 180,E1 -8904.42,E2 -8904.42} C_VEL
LIN {X 0,Y 442.327,Z 444.854,A -85,B 0,C 180,E1 -8904.987,E2 -8904.987} C_VEL
LIN {X 0,Y 441.841,Z 456.082,A -85,B 0,C 180,E1 -8905.667,E2 -8905.667} C_VEL
LIN {X 0,Y 441.174,Z 466.411,A -85,B 0,C 180,E1 -8906.461,E2 -8906.461} C_VEL
LIN {X 0,Y 440.546,Z 477.037,A -85,B 0,C 180,E1 -8907.486,E2 -8907.486} C_VEL
LIN {X 0,Y 440.041,Z 486.599,A -85,B 0,C 180,E1 -8908.628,E2 -8908.628} C_VEL
LIN {X 0,Y 439.628,Z 494.448,A -85,B 0,C 180,E1 -8909.771,E2 -8909.771} C_VEL
LIN {X 0,Y 439.143,Z 502.159,A -85,B 0,C 180,E1 -8911.147,E2 -8911.147} C_VEL
LIN {X 0,Y 438.801,Z 509.229,A -85,B 0,C 180,E1 -8912.754,E2 -8912.754} C_VEL
LIN {X 0,Y 438.574,Z 513.96,A -85,B 0,C 180,E1 -8914.136,E2 -8914.136} C_VEL
LIN {X 0,Y 438.503,Z 517.585,A -85,B 0,C 180,E1 -8915.519,E2 -8915.519} C_VEL
LIN {X 0,Y 438.504,Z 519.461,A -85,B 0,C 180,E1 -8916.442,E2 -8916.442} C_VEL
LIN {X 0,Y 438.328,Z 520.888,A -85,B 0,C 180,E1 -8917.37,E2 -8917.37} C_VEL
LIN {X 0,Y 438.215,Z 522.521,A -85,B 0,C 180,E1 -8919.229,E2 -8919.229} C_VEL
LIN {X 0,Y 438.238,Z 522.749,A -85,B 0,C 180,E1 -8920.161,E2 -8920.161} C_VEL
LIN {X 0,Y 438.269,Z 522.537,A -85,B 0,C 180,E1 -8921.095,E2 -8921.095} C_VEL
LIN {X 0,Y 438.335,Z 521.926,A -85,B 0,C 180,E1 -8922.031,E2 -8922.031} C_VEL
LIN {X 0,Y 438.299,Z 520.92,A -85,B 0,C 180,E1 -8922.973,E2 -8922.973} C_VEL
LIN {X 0,Y 438.38,Z 519.485,A -85,B 0,C 180,E1 -8923.915,E2 -8923.915} C_VEL
LIN {X 0,Y 438.595,Z 516.475,A -85,B 0,C 180,E1 -8925.331,E2 -8925.331} C_VEL
LIN {X 0,Y 438.786,Z 512.358,A -85,B 0,C 180,E1 -8926.757,E2 -8926.757} C_VEL
LIN {X 0,Y 439.2,Z 505.971,A -85,B 0,C 180,E1 -8928.424,E2 -8928.424} C_VEL
LIN {X 0,Y 439.678,Z 498.956,A -85,B 0,C 180,E1 -8929.857,E2 -8929.857} C_VEL
LIN {X 0,Y 440.106,Z 491.72,A -85,B 0,C 180,E1 -8931.057,E2 -8931.057} C_VEL
LIN {X 0,Y 440.798,Z 481.908,A -85,B 0,C 180,E1 -8932.371,E2 -8932.371} C_VEL
LIN {X 0,Y 441.459,Z 471.891,A -85,B 0,C 180,E1 -8933.453,E2 -8933.453} C_VEL
LIN {X 0,Y 442.18,Z 460.853,A -85,B 0,C 180,E1 -8934.409,E2 -8934.409} C_VEL
LIN {X 0,Y 442.78,Z 448.902,A -85,B 0,C 180,E1 -8935.214,E2 -8935.214} C_VEL
LIN {X 0,Y 443.227,Z 436.336,A -85,B 0,C 180,E1 -8935.852,E2 -8935.852} C_VEL
LIN {X 0,Y 443.47,Z 423.351,A -85,B 0,C 180,E1 -8936.311,E2 -8936.311} C_VEL
LIN {X 0,Y 443.836,Z 406.673,A -85,B 0,C 180,E1 -8936.636,E2 -8936.636} C_VEL
LIN {X 0,Y 444.721,Z 329.387,A -85,B 0,C 180,E1 -8937.9,E2 -8937.9} C_VEL
LIN {X 0,Y 440.942,Z 311.74,A -85,B 0,C 180,E1 -8938.41,E2 -8938.41} C_VEL
LIN {X 0,Y 441.071,Z 304.721,A -85,B 0,C 180,E1 -8939.864,E2 -8939.864} C_VEL
LIN {X 0,Y 439.391,Z 295.756,A -85,B 0,C 180,E1 -8941.882,E2 -8941.882} C_VEL
LIN {X 0,Y 439.399,Z 295.751,A -85,B 0,C 180,E1 -8945.156,E2 -8945.156} C_VEL
LIN {X 0,Y 439.377,Z 295.756,A -85,B 0,C 180,E1 -8948.596,E2 -8948.596} C_VEL
LIN {X 0,Y 439.388,Z 295.751,A -85,B 0,C 180,E1 -8951.257,E2 -8951.257} C_VEL
LIN {X 0,Y 439.399,Z 295.753,A -85,B 0,C 180,E1 -8954.73,E2 -8954.73} C_VEL
LIN {X 0,Y 439.395,Z 295.748,A -85,B 0,C 180,E1 -8957.796,E2 -8957.796} C_VEL
LIN {X 0,Y 439.429,Z 295.745,A -85,B 0,C 180,E1 -8960.228,E2 -8960.228} C_VEL
LIN {X 0,Y 439.373,Z 295.749,A -85,B 0,C 180,E1 -8963.713,E2 -8963.713} C_VEL
LIN {X 0,Y 439.372,Z 295.754,A -85,B 0,C 180,E1 -8967.054,E2 -8967.054} C_VEL
LIN {X 0,Y 439.381,Z 295.745,A -85,B 0,C 180,E1 -8970.274,E2 -8970.274} C_VEL
LIN {X 0,Y 439.427,Z 295.745,A -85,B 0,C 180,E1 -8973.396,E2 -8973.396} C_VEL
LIN {X 0,Y 439.385,Z 295.743,A -85,B 0,C 180,E1 -8976.43,E2 -8976.43} C_VEL
LIN {X 0,Y 439.388,Z 295.752,A -85,B 0,C 180,E1 -8979.397,E2 -8979.397} C_VEL
LIN {X 0,Y 439.43,Z 295.744,A -85,B 0,C 180,E1 -8982.31,E2 -8982.31} C_VEL
LIN {X 0,Y 439.447,Z 295.74,A -85,B 0,C 180,E1 -8985.174,E2 -8985.174} C_VEL
LIN {X 0,Y 439.483,Z 295.737,A -85,B 0,C 180,E1 -8988.001,E2 -8988.001} C_VEL
LIN {X 0,Y 439.547,Z 295.736,A -85,B 0,C 180,E1 -8991.726,E2 -8991.726} C_VEL
LIN {X 0,Y 439.616,Z 295.72,A -85,B 0,C 180,E1 -8994.496,E2 -8994.496} C_VEL
LIN {X 0,Y 439.634,Z 295.719,A -85,B 0,C 180,E1 -8998.168,E2 -8998.168} C_VEL
LIN {X 0,Y 439.762,Z 295.708,A -85,B 0,C 180,E1 -9000,E2 -9000} C_VEL
LIN {X 0,Y 439.64,Z 295.714,A -85,B 0,C 180,E1 -9002.749,E2 -9002.749} C_VEL
LIN {X 0,Y 439.612,Z 295.719,A -85,B 0,C 180,E1 -9006.426,E2 -9006.426} C_VEL
LIN {X 0,Y 439.499,Z 295.734,A -85,B 0,C 180,E1 -9009.202,E2 -9009.202} C_VEL
LIN {X 0,Y 439.465,Z 295.74,A -85,B 0,C 180,E1 -9012.938,E2 -9012.938} C_VEL
LIN {X 0,Y 439.447,Z 295.742,A -85,B 0,C 180,E1 -9016.349,E2 -9016.349} C_VEL
LIN {X 0,Y 439.403,Z 295.744,A -85,B 0,C 180,E1 -9019.626,E2 -9019.626} C_VEL
LIN {X 0,Y 439.365,Z 295.757,A -85,B 0,C 180,E1 -9022.576,E2 -9022.576} C_VEL
LIN {X 0,Y 439.405,Z 295.746,A -85,B 0,C 180,E1 -9025.585,E2 -9025.585} C_VEL
LIN {X 0,Y 439.418,Z 295.747,A -85,B 0,C 180,E1 -9028.674,E2 -9028.674} C_VEL
LIN {X 0,Y 439.37,Z 295.749,A -85,B 0,C 180,E1 -9032.031,E2 -9032.031} C_VEL
LIN {X 0,Y 439.395,Z 295.749,A -85,B 0,C 180,E1 -9035.341,E2 -9035.341} C_VEL
LIN {X 0,Y 439.378,Z 295.75,A -85,B 0,C 180,E1 -9038.596,E2 -9038.596} C_VEL
LIN {X 0,Y 439.389,Z 295.742,A -85,B 0,C 180,E1 -9041.257,E2 -9041.257} C_VEL
LIN {X 0,Y 439.401,Z 295.747,A -85,B 0,C 180,E1 -9044.73,E2 -9044.73} C_VEL
LIN {X 0,Y 439.397,Z 295.753,A -85,B 0,C 180,E1 -9047.796,E2 -9047.796} C_VEL
LIN {X 0,Y 439.396,Z 295.749,A -85,B 0,C 180,E1 -9050.224,E2 -9050.224} C_VEL
LIN {X 0,Y 439.376,Z 295.755,A -85,B 0,C 180,E1 -9053.713,E2 -9053.713} C_VEL
LIN {X 0,Y 439.375,Z 295.754,A -85,B 0,C 180,E1 -9057.054,E2 -9057.054} C_VEL
LIN {X 0,Y 439.385,Z 295.755,A -85,B 0,C 180,E1 -9060.274,E2 -9060.274} C_VEL
LIN {X 0,Y 439.492,Z 295.889,A -85,B 0,C 180,E1 -9062.726,E2 -9062.726} C_VEL
LIN {X 0,Y 441.982,Z 307.853,A -85,B 0,C 180,E1 -9065.224,E2 -9065.224} C_VEL
LIN {X 0,Y 442.348,Z 312.3,A -85,B 0,C 180,E1 -9066.1,E2 -9066.1} C_VEL
LIN {X 0,Y 441.225,Z 330.497,A -85,B 0,C 180,E1 -9069.487,E2 -9069.487} C_VEL
LIN {X 0,Y 440.601,Z 342.253,A -85,B 0,C 180,E1 -9071.647,E2 -9071.647} C_VEL
LIN {X 0,Y 444.318,Z 364.817,A -85,B 0,C 180,E1 -9072.209,E2 -9072.209} C_VEL
LIN {X 0,Y 443.581,Z 451.598,A -85,B 0,C 180,E1 -9073.666,E2 -9073.666} C_VEL
LIN {X 0,Y 443.056,Z 464.539,A -85,B 0,C 180,E1 -9074.06,E2 -9074.06} C_VEL
LIN {X 0,Y 442.485,Z 477.085,A -85,B 0,C 180,E1 -9074.63,E2 -9074.63} C_VEL
LIN {X 0,Y 441.811,Z 489.058,A -85,B 0,C 180,E1 -9075.373,E2 -9075.373} C_VEL
LIN {X 0,Y 441.121,Z 500.788,A -85,B 0,C 180,E1 -9076.315,E2 -9076.315} C_VEL
LIN {X 0,Y 440.503,Z 510.862,A -85,B 0,C 180,E1 -9077.328,E2 -9077.328} C_VEL
LIN {X 0,Y 439.875,Z 520.18,A -85,B 0,C 180,E1 -9078.479,E2 -9078.479} C_VEL
LIN {X 0,Y 439.261,Z 529.215,A -85,B 0,C 180,E1 -9079.863,E2 -9079.863} C_VEL
LIN {X 0,Y 438.846,Z 536.515,A -85,B 0,C 180,E1 -9081.249,E2 -9081.249} C_VEL
LIN {X 0,Y 438.581,Z 542.378,A -85,B 0,C 180,E1 -9082.634,E2 -9082.634} C_VEL
LIN {X 0,Y 438.371,Z 546.935,A -85,B 0,C 180,E1 -9083.996,E2 -9083.996} C_VEL
LIN {X 0,Y 438.342,Z 550.534,A -85,B 0,C 180,E1 -9085.402,E2 -9085.402} C_VEL
LIN {X 0,Y 438.282,Z 552.325,A -85,B 0,C 180,E1 -9086.322,E2 -9086.322} C_VEL
LIN {X 0,Y 438.341,Z 553.687,A -85,B 0,C 180,E1 -9087.243,E2 -9087.243} C_VEL
LIN {X 0,Y 438.295,Z 554.651,A -85,B 0,C 180,E1 -9088.162,E2 -9088.162} C_VEL
LIN {X 0,Y 438.254,Z 555.227,A -85,B 0,C 180,E1 -9089.081,E2 -9089.081} C_VEL
LIN {X 0,Y 438.281,Z 555.382,A -85,B 0,C 180,E1 -9090,E2 -9090} C_VEL
LIN {X 0,Y 438.295,Z 554.484,A -85,B 0,C 180,E1 -9091.837,E2 -9091.837} C_VEL
LIN {X 0,Y 438.359,Z 553.453,A -85,B 0,C 180,E1 -9092.756,E2 -9092.756} C_VEL
LIN {X 0,Y 438.285,Z 551.979,A -85,B 0,C 180,E1 -9093.677,E2 -9093.677} C_VEL
LIN {X 0,Y 438.383,Z 548.964,A -85,B 0,C 180,E1 -9095.058,E2 -9095.058} C_VEL
LIN {X 0,Y 438.448,Z 544.882,A -85,B 0,C 180,E1 -9096.442,E2 -9096.442} C_VEL
LIN {X 0,Y 438.669,Z 538.605,A -85,B 0,C 180,E1 -9098.058,E2 -9098.058} C_VEL
LIN {X 0,Y 438.973,Z 531.766,A -85,B 0,C 180,E1 -9099.445,E2 -9099.445} C_VEL
LIN {X 0,Y 439.414,Z 523.248,A -85,B 0,C 180,E1 -9100.832,E2 -9100.832} C_VEL
LIN {X 0,Y 439.969,Z 514.475,A -85,B 0,C 180,E1 -9101.985,E2 -9101.985} C_VEL
LIN {X 0,Y 440.574,Z 503.398,A -85,B 0,C 180,E1 -9103.165,E2 -9103.165} C_VEL
LIN {X 0,Y 441.127,Z 492.873,A -85,B 0,C 180,E1 -9104.061,E2 -9104.061} C_VEL
LIN {X 0,Y 441.76,Z 480.752,A -85,B 0,C 180,E1 -9104.864,E2 -9104.864} C_VEL
LIN {X 0,Y 442.281,Z 468.091,A -85,B 0,C 180,E1 -9105.495,E2 -9105.495} C_VEL
LIN {X 0,Y 442.768,Z 455.796,A -85,B 0,C 180,E1 -9105.92,E2 -9105.92} C_VEL
LIN {X 0,Y 443.05,Z 440.134,A -85,B 0,C 180,E1 -9106.235,E2 -9106.235} C_VEL
LIN {X 0,Y 443.615,Z 364.999,A -85,B 0,C 180,E1 -9107.452,E2 -9107.452} C_VEL
LIN {X 0,Y 440.276,Z 342.54,A -85,B 0,C 180,E1 -9107.944,E2 -9107.944} C_VEL
LIN {X 0,Y 441.25,Z 322.989,A -85,B 0,C 180,E1 -9111.489,E2 -9111.489} C_VEL
LIN {X 0,Y 441.929,Z 309.705,A -85,B 0,C 180,E1 -9113.924,E2 -9113.924} C_VEL
LIN {X 0,Y 440.386,Z 300.238,A -85,B 0,C 180,E1 -9115.775,E2 -9115.775} C_VEL
LIN {X 0,Y 439.458,Z 295.743,A -85,B 0,C 180,E1 -9116.697,E2 -9116.697} C_VEL
LIN {X 0,Y 439.382,Z 295.754,A -85,B 0,C 180,E1 -9119.725,E2 -9119.725} C_VEL
LIN {X 0,Y 439.372,Z 295.75,A -85,B 0,C 180,E1 -9122.945,E2 -9122.945} C_VEL
LIN {X 0,Y 439.373,Z 295.758,A -85,B 0,C 180,E1 -9126.287,E2 -9126.287} C_VEL
LIN {X 0,Y 439.4,Z 295.748,A -85,B 0,C 180,E1 -9129.848,E2 -9129.848} C_VEL
LIN {X 0,Y 439.38,Z 295.755,A -85,B 0,C 180,E1 -9132.626,E2 -9132.626} C_VEL
LIN {X 0,Y 439.397,Z 295.747,A -85,B 0,C 180,E1 -9135.27,E2 -9135.27} C_VEL
LIN {X 0,Y 439.386,Z 295.755,A -85,B 0,C 180,E1 -9138.743,E2 -9138.743} C_VEL
LIN {X 0,Y 439.373,Z 295.75,A -85,B 0,C 180,E1 -9141.607,E2 -9141.607} C_VEL
LIN {X 0,Y 439.396,Z 295.754,A -85,B 0,C 180,E1 -9144.843,E2 -9144.843} C_VEL
LIN {X 0,Y 439.369,Z 295.751,A -85,B 0,C 180,E1 -9148.139,E2 -9148.139} C_VEL
LIN {X 0,Y 439.429,Z 295.744,A -85,B 0,C 180,E1 -9151.598,E2 -9151.598} C_VEL
LIN {X 0,Y 439.401,Z 295.747,A -85,B 0,C 180,E1 -9154.415,E2 -9154.415} C_VEL
LIN {X 0,Y 439.361,Z 295.755,A -85,B 0,C 180,E1 -9157.424,E2 -9157.424} C_VEL
LIN {X 0,Y 439.437,Z 295.744,A -85,B 0,C 180,E1 -9160.662,E2 -9160.662} C_VEL
LIN {X 0,Y 439.458,Z 295.739,A -85,B 0,C 180,E1 -9164.224,E2 -9164.224} C_VEL
LIN {X 0,Y 439.479,Z 295.738,A -85,B 0,C 180,E1 -9168.001,E2 -9168.001} C_VEL
LIN {X 0,Y 439.543,Z 295.734,A -85,B 0,C 180,E1 -9171.726,E2 -9171.726} C_VEL
LIN {X 0,Y 439.614,Z 295.72,A -85,B 0,C 180,E1 -9174.495,E2 -9174.495} C_VEL
LIN {X 0,Y 439.628,Z 295.72,A -85,B 0,C 180,E1 -9178.168,E2 -9178.168} C_VEL
LIN {X 0,Y 439.756,Z 295.707,A -85,B 0,C 180,E1 -9180,E2 -9180} C_VEL
LIN {X 0,Y 439.636,Z 295.717,A -85,B 0,C 180,E1 -9182.749,E2 -9182.749} C_VEL
LIN {X 0,Y 439.586,Z 295.725,A -85,B 0,C 180,E1 -9186.425,E2 -9186.425} C_VEL
LIN {X 0,Y 439.494,Z 295.735,A -85,B 0,C 180,E1 -9189.202,E2 -9189.202} C_VEL
LIN {X 0,Y 439.46,Z 295.739,A -85,B 0,C 180,E1 -9192.938,E2 -9192.938} C_VEL
LIN {X 0,Y 439.44,Z 295.747,A -85,B 0,C 180,E1 -9196.348,E2 -9196.348} C_VEL
LIN {X 0,Y 439.396,Z 295.748,A -85,B 0,C 180,E1 -9199.626,E2 -9199.626} C_VEL
LIN {X 0,Y 439.358,Z 295.757,A -85,B 0,C 180,E1 -9202.576,E2 -9202.576} C_VEL
LIN {X 0,Y 439.383,Z 295.749,A -85,B 0,C 180,E1 -9205.586,E2 -9205.586} C_VEL
LIN {X 0,Y 439.411,Z 295.751,A -85,B 0,C 180,E1 -9208.674,E2 -9208.674} C_VEL
LIN {X 0,Y 439.364,Z 295.752,A -85,B 0,C 180,E1 -9212.031,E2 -9212.031} C_VEL
LIN {X 0,Y 439.389,Z 295.749,A -85,B 0,C 180,E1 -9215.341,E2 -9215.341} C_VEL
LIN {X 0,Y 439.372,Z 295.756,A -85,B 0,C 180,E1 -9218.596,E2 -9218.596} C_VEL
LIN {X 0,Y 439.384,Z 295.751,A -85,B 0,C 180,E1 -9221.257,E2 -9221.257} C_VEL
LIN {X 0,Y 439.396,Z 295.752,A -85,B 0,C 180,E1 -9224.73,E2 -9224.73} C_VEL
LIN {X 0,Y 439.354,Z 295.753,A -85,B 0,C 180,E1 -9227.792,E2 -9227.792} C_VEL
LIN {X 0,Y 439.354,Z 295.752,A -85,B 0,C 180,E1 -9230.22,E2 -9230.22} C_VEL
LIN {X 0,Y 439.369,Z 295.752,A -85,B 0,C 180,E1 -9233.713,E2 -9233.713} C_VEL
LIN {X 0,Y 439.369,Z 295.755,A -85,B 0,C 180,E1 -9237.054,E2 -9237.054} C_VEL
LIN {X 0,Y 439.368,Z 295.75,A -85,B 0,C 180,E1 -9240.274,E2 -9240.274} C_VEL
LIN {X 0,Y 439.362,Z 295.759,A -85,B 0,C 180,E1 -9243.392,E2 -9243.392} C_VEL
LIN {X 0,Y 439.363,Z 295.751,A -85,B 0,C 180,E1 -9246.429,E2 -9246.429} C_VEL
LIN {X 0,Y 439.386,Z 295.753,A -85,B 0,C 180,E1 -9249.398,E2 -9249.398} C_VEL
LIN {X 0,Y 439.4,Z 295.748,A -85,B 0,C 180,E1 -9252.309,E2 -9252.309} C_VEL
LIN {X 0,Y 439.445,Z 295.742,A -85,B 0,C 180,E1 -9255.174,E2 -9255.174} C_VEL
LIN {X 0,Y 439.462,Z 295.746,A -85,B 0,C 180,E1 -9258.469,E2 -9258.469} C_VEL
LIN {X 0,Y 439.496,Z 295.932,A -85,B 0,C 180,E1 -9258.762,E2 -9258.762} C_VEL
LIN {X 0,Y 440.751,Z 304.35,A -85,B 0,C 180,E1 -9260.594,E2 -9260.594} C_VEL
LIN {X 0,Y 440.551,Z 311.918,A -85,B 0,C 180,E1 -9262.138,E2 -9262.138} C_VEL
LIN {X 0,Y 443.878,Z 329.58,A -85,B 0,C 180,E1 -9262.553,E2 -9262.553} C_VEL
LIN {X 0,Y 443.596,Z 364.832,A -85,B 0,C 180,E1 -9263.125,E2 -9263.125} C_VEL
LIN {X 0,Y 442.878,Z 370.675,A -85,B 0,C 180,E1 -9263.197,E2 -9263.197} C_VEL
LIN {X 0,Y 437.1,Z 389.646,A -85,B 0,C 180,E1 -9263.312,E2 -9263.312} C_VEL
LIN {X 0,Y 436.385,Z 395.489,A -85,B 0,C 180,E1 -9263.385,E2 -9263.385} C_VEL
LIN {X 0,Y 436.087,Z 421.114,A -85,B 0,C 180,E1 -9263.842,E2 -9263.842} C_VEL
LIN {X 0,Y 435.73,Z 434.407,A -85,B 0,C 180,E1 -9264.273,E2 -9264.273} C_VEL
LIN {X 0,Y 435.371,Z 446.425,A -85,B 0,C 180,E1 -9264.849,E2 -9264.849} C_VEL
LIN {X 0,Y 434.846,Z 458.093,A -85,B 0,C 180,E1 -9265.597,E2 -9265.597} C_VEL
LIN {X 0,Y 434.058,Z 469.384,A -85,B 0,C 180,E1 -9266.519,E2 -9266.519} C_VEL
LIN {X 0,Y 433.403,Z 479.546,A -85,B 0,C 180,E1 -9267.561,E2 -9267.561} C_VEL
LIN {X 0,Y 432.941,Z 489.456,A -85,B 0,C 180,E1 -9268.838,E2 -9268.838} C_VEL
LIN {X 0,Y 432.418,Z 498.205,A -85,B 0,C 180,E1 -9270.233,E2 -9270.233} C_VEL
LIN {X 0,Y 431.94,Z 505.242,A -85,B 0,C 180,E1 -9271.632,E2 -9271.632} C_VEL
LIN {X 0,Y 431.639,Z 511.653,A -85,B 0,C 180,E1 -9273.267,E2 -9273.267} C_VEL
LIN {X 0,Y 431.393,Z 515.904,A -85,B 0,C 180,E1 -9274.673,E2 -9274.673} C_VEL
LIN {X 0,Y 431.42,Z 519.751,A -85,B 0,C 180,E1 -9276.429,E2 -9276.429} C_VEL
LIN {X 0,Y 431.238,Z 521.313,A -85,B 0,C 180,E1 -9277.492,E2 -9277.492} C_VEL
LIN {X 0,Y 431.118,Z 522.855,A -85,B 0,C 180,E1 -9279.382,E2 -9279.382} C_VEL
LIN {X 0,Y 431.145,Z 523,A -85,B 0,C 180,E1 -9280.33,E2 -9280.33} C_VEL
LIN {X 0,Y 431.253,Z 522.191,A -85,B 0,C 180,E1 -9282.095,E2 -9282.095} C_VEL
LIN {X 0,Y 431.234,Z 521.021,A -85,B 0,C 180,E1 -9283.189,E2 -9283.189} C_VEL
LIN {X 0,Y 431.317,Z 519.494,A -85,B 0,C 180,E1 -9284.147,E2 -9284.147} C_VEL
LIN {X 0,Y 431.544,Z 516.384,A -85,B 0,C 180,E1 -9285.588,E2 -9285.588} C_VEL
LIN {X 0,Y 431.783,Z 512.158,A -85,B 0,C 180,E1 -9287.037,E2 -9287.037} C_VEL
LIN {X 0,Y 432.25,Z 505.656,A -85,B 0,C 180,E1 -9288.731,E2 -9288.731} C_VEL
LIN {X 0,Y 432.78,Z 498.475,A -85,B 0,C 180,E1 -9290.187,E2 -9290.187} C_VEL
LIN {X 0,Y 433.379,Z 489.395,A -85,B 0,C 180,E1 -9291.65,E2 -9291.65} C_VEL
LIN {X 0,Y 434.12,Z 480.022,A -85,B 0,C 180,E1 -9292.864,E2 -9292.864} C_VEL
LIN {X 0,Y 434.789,Z 469.47,A -85,B 0,C 180,E1 -9293.962,E2 -9293.962} C_VEL
LIN {X 0,Y 435.557,Z 458.215,A -85,B 0,C 180,E1 -9294.89,E2 -9294.89} C_VEL
LIN {X 0,Y 436.126,Z 446.365,A -85,B 0,C 180,E1 -9295.658,E2 -9295.658} C_VEL
LIN {X 0,Y 436.626,Z 433.307,A -85,B 0,C 180,E1 -9296.273,E2 -9296.273} C_VEL
LIN {X 0,Y 436.833,Z 420.784,A -85,B 0,C 180,E1 -9296.678,E2 -9296.678} C_VEL
LIN {X 0,Y 437.274,Z 394.454,A -85,B 0,C 180,E1 -9297.143,E2 -9297.143} C_VEL
LIN {X 0,Y 438.138,Z 330.824,A -85,B 0,C 180,E1 -9298.195,E2 -9298.195} C_VEL
LIN {X 0,Y 434.065,Z 312.017,A -85,B 0,C 180,E1 -9298.749,E2 -9298.749} C_VEL
LIN {X 0,Y 434.109,Z 305.505,A -85,B 0,C 180,E1 -9300.124,E2 -9300.124} C_VEL
LIN {X 0,Y 432.34,Z 296.633,A -85,B 0,C 180,E1 -9302.166,E2 -9302.166} C_VEL
LIN {X 0,Y 432.339,Z 296.634,A -85,B 0,C 180,E1 -9304.677,E2 -9304.677} C_VEL
LIN {X 0,Y 432.336,Z 296.626,A -85,B 0,C 180,E1 -9308.15,E2 -9308.15} C_VEL
LIN {X 0,Y 432.332,Z 296.629,A -85,B 0,C 180,E1 -9311.602,E2 -9311.602} C_VEL
LIN {X 0,Y 432.333,Z 296.631,A -85,B 0,C 180,E1 -9314.347,E2 -9314.347} C_VEL
LIN {X 0,Y 432.319,Z 296.633,A -85,B 0,C 180,E1 -9317.016,E2 -9317.016} C_VEL
LIN {X 0,Y 432.335,Z 296.627,A -85,B 0,C 180,E1 -9319.82,E2 -9319.82} C_VEL
LIN {X 0,Y 432.306,Z 296.634,A -85,B 0,C 180,E1 -9323.022,E2 -9323.022} C_VEL
LIN {X 0,Y 432.358,Z 296.621,A -85,B 0,C 180,E1 -9325.997,E2 -9325.997} C_VEL
LIN {X 0,Y 432.346,Z 296.625,A -85,B 0,C 180,E1 -9329.49,E2 -9329.49} C_VEL
LIN {X 0,Y 432.39,Z 296.618,A -85,B 0,C 180,E1 -9332.928,E2 -9332.928} C_VEL
LIN {X 0,Y 432.369,Z 296.617,A -85,B 0,C 180,E1 -9336.023,E2 -9336.023} C_VEL
LIN {X 0,Y 432.35,Z 296.628,A -85,B 0,C 180,E1 -9339.046,E2 -9339.046} C_VEL
LIN {X 0,Y 432.377,Z 296.624,A -85,B 0,C 180,E1 -9342.011,E2 -9342.011} C_VEL
LIN {X 0,Y 432.394,Z 296.617,A -85,B 0,C 180,E1 -9344.927,E2 -9344.927} C_VEL
LIN {X 0,Y 432.458,Z 296.615,A -85,B 0,C 180,E1 -9347.804,E2 -9347.804} C_VEL
LIN {X 0,Y 432.491,Z 296.613,A -85,B 0,C 180,E1 -9351.591,E2 -9351.591} C_VEL
LIN {X 0,Y 432.592,Z 296.596,A -85,B 0,C 180,E1 -9354.406,E2 -9354.406} C_VEL
LIN {X 0,Y 432.603,Z 296.595,A -85,B 0,C 180,E1 -9358.138,E2 -9358.138} C_VEL
LIN {X 0,Y 432.731,Z 296.583,A -85,B 0,C 180,E1 -9360,E2 -9360} C_VEL
LIN {X 0,Y 432.592,Z 296.591,A -85,B 0,C 180,E1 -9362.794,E2 -9362.794} C_VEL
LIN {X 0,Y 432.568,Z 296.595,A -85,B 0,C 180,E1 -9366.531,E2 -9366.531} C_VEL
LIN {X 0,Y 432.442,Z 296.613,A -85,B 0,C 180,E1 -9369.353,E2 -9369.353} C_VEL
LIN {X 0,Y 432.431,Z 296.617,A -85,B 0,C 180,E1 -9372.804,E2 -9372.804} C_VEL
LIN {X 0,Y 432.413,Z 296.618,A -85,B 0,C 180,E1 -9376.479,E2 -9376.479} C_VEL
LIN {X 0,Y 432.339,Z 296.625,A -85,B 0,C 180,E1 -9379.961,E2 -9379.961} C_VEL
LIN {X 0,Y 432.319,Z 296.633,A -85,B 0,C 180,E1 -9382.964,E2 -9382.964} C_VEL
LIN {X 0,Y 432.365,Z 296.623,A -85,B 0,C 180,E1 -9386.033,E2 -9386.033} C_VEL
LIN {X 0,Y 432.343,Z 296.63,A -85,B 0,C 180,E1 -9389.188,E2 -9389.188} C_VEL
LIN {X 0,Y 432.324,Z 296.628,A -85,B 0,C 180,E1 -9392.443,E2 -9392.443} C_VEL
LIN {X 0,Y 432.345,Z 296.625,A -85,B 0,C 180,E1 -9395.632,E2 -9395.632} C_VEL
LIN {X 0,Y 432.341,Z 296.628,A -85,B 0,C 180,E1 -9398.715,E2 -9398.715} C_VEL
LIN {X 0,Y 432.335,Z 296.629,A -85,B 0,C 180,E1 -9401.797,E2 -9401.797} C_VEL
LIN {X 0,Y 432.335,Z 296.626,A -85,B 0,C 180,E1 -9404.348,E2 -9404.348} C_VEL
LIN {X 0,Y 432.321,Z 296.632,A -85,B 0,C 180,E1 -9407.016,E2 -9407.016} C_VEL
LIN {X 0,Y 432.335,Z 296.632,A -85,B 0,C 180,E1 -9409.821,E2 -9409.821} C_VEL
LIN {X 0,Y 432.308,Z 296.629,A -85,B 0,C 180,E1 -9413.022,E2 -9413.022} C_VEL
LIN {X 0,Y 432.361,Z 296.629,A -85,B 0,C 180,E1 -9415.997,E2 -9415.997} C_VEL
LIN {X 0,Y 432.35,Z 296.629,A -85,B 0,C 180,E1 -9419.49,E2 -9419.49} C_VEL
LIN {X 0,Y 432.422,Z 296.674,A -85,B 0,C 180,E1 -9422.406,E2 -9422.406} C_VEL
LIN {X 0,Y 434.833,Z 308.066,A -85,B 0,C 180,E1 -9424.838,E2 -9424.838} C_VEL
LIN {X 0,Y 435.467,Z 313.56,A -85,B 0,C 180,E1 -9425.951,E2 -9425.951} C_VEL
LIN {X 0,Y 434.286,Z 331.613,A -85,B 0,C 180,E1 -9429.367,E2 -9429.367} C_VEL
LIN {X 0,Y 433.723,Z 342,A -85,B 0,C 180,E1 -9431.308,E2 -9431.308} C_VEL
LIN {X 0,Y 437.389,Z 364.063,A -85,B 0,C 180,E1 -9431.87,E2 -9431.87} C_VEL
LIN {X 0,Y 437.795,Z 369.031,A -85,B 0,C 180,E1 -9431.975,E2 -9431.975} C_VEL
LIN {X 0,Y 436.872,Z 450.44,A -85,B 0,C 180,E1 -9433.348,E2 -9433.348} C_VEL
LIN {X 0,Y 436.347,Z 463.673,A -85,B 0,C 180,E1 -9433.749,E2 -9433.749} C_VEL
LIN {X 0,Y 435.74,Z 476.368,A -85,B 0,C 180,E1 -9434.326,E2 -9434.326} C_VEL
LIN {X 0,Y 435.035,Z 487.675,A -85,B 0,C 180,E1 -9435.02,E2 -9435.02} C_VEL
LIN {X 0,Y 434.283,Z 499.338,A -85,B 0,C 180,E1 -9435.951,E2 -9435.951} C_VEL
LIN {X 0,Y 433.615,Z 509.834,A -85,B 0,C 180,E1 -9437.004,E2 -9437.004} C_VEL
LIN {X 0,Y 433.039,Z 518.429,A -85,B 0,C 180,E1 -9438.058,E2 -9438.058} C_VEL
LIN {X 0,Y 432.389,Z 526.367,A -85,B 0,C 180,E1 -9439.227,E2 -9439.227} C_VEL
LIN {X 0,Y 431.921,Z 534.16,A -85,B 0,C 180,E1 -9440.635,E2 -9440.635} C_VEL
LIN {X 0,Y 431.576,Z 540.413,A -85,B 0,C 180,E1 -9442.043,E2 -9442.043} C_VEL
LIN {X 0,Y 431.327,Z 546.115,A -85,B 0,C 180,E1 -9443.685,E2 -9443.685} C_VEL
LIN {X 0,Y 431.271,Z 550.337,A -85,B 0,C 180,E1 -9445.326,E2 -9445.326} C_VEL
LIN {X 0,Y 431.188,Z 552.106,A -85,B 0,C 180,E1 -9446.262,E2 -9446.262} C_VEL
LIN {X 0,Y 431.237,Z 553.457,A -85,B 0,C 180,E1 -9447.197,E2 -9447.197} C_VEL
LIN {X 0,Y 431.219,Z 554.412,A -85,B 0,C 180,E1 -9448.132,E2 -9448.132} C_VEL
LIN {X 0,Y 431.171,Z 554.977,A -85,B 0,C 180,E1 -9449.066,E2 -9449.066} C_VEL
LIN {X 0,Y 431.193,Z 555.112,A -85,B 0,C 180,E1 -9450,E2 -9450} C_VEL
LIN {X 0,Y 431.219,Z 554.195,A -85,B 0,C 180,E1 -9451.868,E2 -9451.868} C_VEL
LIN {X 0,Y 431.268,Z 553.152,A -85,B 0,C 180,E1 -9452.802,E2 -9452.802} C_VEL
LIN {X 0,Y 431.192,Z 551.656,A -85,B 0,C 180,E1 -9453.738,E2 -9453.738} C_VEL
LIN {X 0,Y 431.293,Z 548.619,A -85,B 0,C 180,E1 -9455.142,E2 -9455.142} C_VEL
LIN {X 0,Y 431.376,Z 544.511,A -85,B 0,C 180,E1 -9456.548,E2 -9456.548} C_VEL
LIN {X 0,Y 431.602,Z 538.205,A -85,B 0,C 180,E1 -9458.191,E2 -9458.191} C_VEL
LIN {X 0,Y 431.916,Z 531.332,A -85,B 0,C 180,E1 -9459.6,E2 -9459.6} C_VEL
LIN {X 0,Y 432.415,Z 522.758,A -85,B 0,C 180,E1 -9461.009,E2 -9461.009} C_VEL
LIN {X 0,Y 432.967,Z 513.934,A -85,B 0,C 180,E1 -9462.182,E2 -9462.182} C_VEL
LIN {X 0,Y 433.56,Z 503.811,A -85,B 0,C 180,E1 -9463.28,E2 -9463.28} C_VEL
LIN {X 0,Y 434.106,Z 493.653,A -85,B 0,C 180,E1 -9464.174,E2 -9464.174} C_VEL
LIN {X 0,Y 434.769,Z 481.914,A -85,B 0,C 180,E1 -9464.989,E2 -9464.989} C_VEL
LIN {X 0,Y 435.332,Z 469.69,A -85,B 0,C 180,E1 -9465.628,E2 -9465.628} C_VEL
LIN {X 0,Y 435.786,Z 457.265,A -85,B 0,C 180,E1 -9466.092,E2 -9466.092} C_VEL
LIN {X 0,Y 436.127,Z 444.929,A -85,B 0,C 180,E1 -9466.379,E2 -9466.379} C_VEL
LIN {X 0,Y 436.751,Z 365.709,A -85,B 0,C 180,E1 -9467.683,E2 -9467.683} C_VEL
LIN {X 0,Y 433.319,Z 342.198,A -85,B 0,C 180,E1 -9468.219,E2 -9468.219} C_VEL
LIN {X 0,Y 434.269,Z 323.83,A -85,B 0,C 180,E1 -9471.603,E2 -9471.603} C_VEL
LIN {X 0,Y 434.961,Z 310.54,A -85,B 0,C 180,E1 -9474.078,E2 -9474.078} C_VEL
LIN {X 0,Y 433.309,Z 301.041,A -85,B 0,C 180,E1 -9475.971,E2 -9475.971} C_VEL
LIN {X 0,Y 432.428,Z 296.619,A -85,B 0,C 180,E1 -9476.874,E2 -9476.874} C_VEL
LIN {X 0,Y 432.345,Z 296.634,A -85,B 0,C 180,E1 -9480.259,E2 -9480.259} C_VEL
LIN {X 0,Y 432.339,Z 296.627,A -85,B 0,C 180,E1 -9483.551,E2 -9483.551} C_VEL
LIN {X 0,Y 432.337,Z 296.629,A -85,B 0,C 180,E1 -9485.817,E2 -9485.817} C_VEL
LIN {X 0,Y 432.326,Z 296.628,A -85,B 0,C 180,E1 -9489.345,E2 -9489.345} C_VEL
LIN {X 0,Y 432.331,Z 296.628,A -85,B 0,C 180,E1 -9491.796,E2 -9491.796} C_VEL
LIN {X 0,Y 432.331,Z 296.633,A -85,B 0,C 180,E1 -9494.347,E2 -9494.347} C_VEL
LIN {X 0,Y 432.318,Z 296.631,A -85,B 0,C 180,E1 -9497.015,E2 -9497.015} C_VEL
LIN {X 0,Y 432.333,Z 296.627,A -85,B 0,C 180,E1 -9499.82,E2 -9499.82} C_VEL
LIN {X 0,Y 432.304,Z 296.635,A -85,B 0,C 180,E1 -9503.021,E2 -9503.021} C_VEL
LIN {X 0,Y 432.356,Z 296.624,A -85,B 0,C 180,E1 -9505.996,E2 -9505.996} C_VEL
LIN {X 0,Y 432.344,Z 296.627,A -85,B 0,C 180,E1 -9509.489,E2 -9509.489} C_VEL
LIN {X 0,Y 432.387,Z 296.628,A -85,B 0,C 180,E1 -9512.928,E2 -9512.928} C_VEL
LIN {X 0,Y 432.367,Z 296.622,A -85,B 0,C 180,E1 -9516.023,E2 -9516.023} C_VEL
LIN {X 0,Y 432.346,Z 296.632,A -85,B 0,C 180,E1 -9519.046,E2 -9519.046} C_VEL
LIN {X 0,Y 432.373,Z 296.622,A -85,B 0,C 180,E1 -9522.011,E2 -9522.011} C_VEL
LIN {X 0,Y 432.392,Z 296.623,A -85,B 0,C 180,E1 -9524.926,E2 -9524.926} C_VEL
LIN {X 0,Y 432.454,Z 296.615,A -85,B 0,C 180,E1 -9527.803,E2 -9527.803} C_VEL
LIN {X 0,Y 432.487,Z 296.615,A -85,B 0,C 180,E1 -9531.59,E2 -9531.59} C_VEL
LIN {X 0,Y 432.591,Z 296.595,A -85,B 0,C 180,E1 -9534.406,E2 -9534.406} C_VEL
LIN {X 0,Y 432.598,Z 296.596,A -85,B 0,C 180,E1 -9538.138,E2 -9538.138} C_VEL
LIN {X 0,Y 432.726,Z 296.582,A -85,B 0,C 180,E1 -9540,E2 -9540} C_VEL
LIN {X 0,Y 432.588,Z 296.595,A -85,B 0,C 180,E1 -9542.793,E2 -9542.793} C_VEL
LIN {X 0,Y 432.58,Z 296.6,A -85,B 0,C 180,E1 -9545.594,E2 -9545.594} C_VEL
LIN {X 0,Y 432.477,Z 296.611,A -85,B 0,C 180,E1 -9548.41,E2 -9548.41} C_VEL
LIN {X 0,Y 432.454,Z 296.618,A -85,B 0,C 180,E1 -9552.197,E2 -9552.197} C_VEL
LIN {X 0,Y 432.424,Z 296.622,A -85,B 0,C 180,E1 -9556.039,E2 -9556.039} C_VEL
LIN {X 0,Y 432.381,Z 296.621,A -85,B 0,C 180,E1 -9559.485,E2 -9559.485} C_VEL
LIN {X 0,Y 432.312,Z 296.631,A -85,B 0,C 180,E1 -9562.964,E2 -9562.964} C_VEL
LIN {X 0,Y 432.337,Z 296.628,A -85,B 0,C 180,E1 -9565.002,E2 -9565.002} C_VEL
LIN {X 0,Y 432.375,Z 296.625,A -85,B 0,C 180,E1 -9568.124,E2 -9568.124} C_VEL
LIN {X 0,Y 432.316,Z 296.629,A -85,B 0,C 180,E1 -9571.346,E2 -9571.346} C_VEL
LIN {X 0,Y 432.335,Z 296.635,A -85,B 0,C 180,E1 -9574.677,E2 -9574.677} C_VEL
LIN {X 0,Y 432.331,Z 296.628,A -85,B 0,C 180,E1 -9578.15,E2 -9578.15} C_VEL
LIN {X 0,Y 432.328,Z 296.628,A -85,B 0,C 180,E1 -9581.602,E2 -9581.602} C_VEL
LIN {X 0,Y 432.329,Z 296.629,A -85,B 0,C 180,E1 -9584.348,E2 -9584.348} C_VEL
LIN {X 0,Y 432.302,Z 296.639,A -85,B 0,C 180,E1 -9587.018,E2 -9587.018} C_VEL
LIN {X 0,Y 432.304,Z 296.631,A -85,B 0,C 180,E1 -9589.825,E2 -9589.825} C_VEL
LIN {X 0,Y 432.302,Z 296.637,A -85,B 0,C 180,E1 -9593.022,E2 -9593.022} C_VEL
LIN {X 0,Y 432.354,Z 296.625,A -85,B 0,C 180,E1 -9595.997,E2 -9595.997} C_VEL
LIN {X 0,Y 432.343,Z 296.632,A -85,B 0,C 180,E1 -9599.491,E2 -9599.491} C_VEL
LIN {X 0,Y 432.324,Z 296.63,A -85,B 0,C 180,E1 -9601.873,E2 -9601.873} C_VEL
LIN {X 0,Y 432.347,Z 296.633,A -85,B 0,C 180,E1 -9605.547,E2 -9605.547} C_VEL
LIN {X 0,Y 432.348,Z 296.626,A -85,B 0,C 180,E1 -9609.047,E2 -9609.047} C_VEL
LIN {X 0,Y 432.356,Z 296.628,A -85,B 0,C 180,E1 -9612.011,E2 -9612.011} C_VEL
LIN {X 0,Y 432.392,Z 296.619,A -85,B 0,C 180,E1 -9614.927,E2 -9614.927} C_VEL
LIN {X 0,Y 432.437,Z 296.621,A -85,B 0,C 180,E1 -9618.279,E2 -9618.279} C_VEL
LIN {X 0,Y 432.452,Z 296.753,A -85,B 0,C 180,E1 -9618.577,E2 -9618.577} C_VEL
LIN {X 0,Y 433.761,Z 305.183,A -85,B 0,C 180,E1 -9620.441,E2 -9620.441} C_VEL
LIN {X 0,Y 433.578,Z 312.034,A -85,B 0,C 180,E1 -9621.873,E2 -9621.873} C_VEL
LIN {X 0,Y 437.044,Z 330.704,A -85,B 0,C 180,E1 -9622.322,E2 -9622.322} C_VEL
LIN {X 0,Y 436.385,Z 395.489,A -85,B 0,C 180,E1 -9623.385,E2 -9623.385} C_VEL
LIN {X 0,Y 435.675,Z 401.342,A -85,B 0,C 180,E1 -9623.453,E2 -9623.453} C_VEL
LIN {X 0,Y 429.871,Z 420.284,A -85,B 0,C 180,E1 -9623.602,E2 -9623.602} C_VEL
LIN {X 0,Y 429.1,Z 426.036,A -85,B 0,C 180,E1 -9623.744,E2 -9623.744} C_VEL
LIN {X 0,Y 428.737,Z 438.886,A -85,B 0,C 180,E1 -9624.238,E2 -9624.238} C_VEL
LIN {X 0,Y 428.344,Z 449.822,A -85,B 0,C 180,E1 -9624.823,E2 -9624.823} C_VEL
LIN {X 0,Y 427.78,Z 461.61,A -85,B 0,C 180,E1 -9625.643,E2 -9625.643} C_VEL
LIN {X 0,Y 427.052,Z 471.033,A -85,B 0,C 180,E1 -9626.462,E2 -9626.462} C_VEL
LIN {X 0,Y 426.427,Z 479.912,A -85,B 0,C 180,E1 -9627.403,E2 -9627.403} C_VEL
LIN {X 0,Y 425.964,Z 489,A -85,B 0,C 180,E1 -9628.582,E2 -9628.582} C_VEL
LIN {X 0,Y 425.415,Z 497.869,A -85,B 0,C 180,E1 -9630,E2 -9630} C_VEL
LIN {X 0,Y 424.917,Z 505.034,A -85,B 0,C 180,E1 -9631.422,E2 -9631.422} C_VEL
LIN {X 0,Y 424.634,Z 510.754,A -85,B 0,C 180,E1 -9632.846,E2 -9632.846} C_VEL
LIN {X 0,Y 424.36,Z 515.272,A -85,B 0,C 180,E1 -9634.274,E2 -9634.274} C_VEL
LIN {X 0,Y 424.337,Z 518.702,A -85,B 0,C 180,E1 -9635.703,E2 -9635.703} C_VEL
LIN {X 0,Y 424.284,Z 520.418,A -85,B 0,C 180,E1 -9636.659,E2 -9636.659} C_VEL
LIN {X 0,Y 424.066,Z 522.656,A -85,B 0,C 180,E1 -9638.578,E2 -9638.578} C_VEL
LIN {X 0,Y 424.021,Z 523.165,A -85,B 0,C 180,E1 -9639.541,E2 -9639.541} C_VEL
LIN {X 0,Y 424.062,Z 523.243,A -85,B 0,C 180,E1 -9640.504,E2 -9640.504} C_VEL
LIN {X 0,Y 424.159,Z 522.466,A -85,B 0,C 180,E1 -9642.154,E2 -9642.154} C_VEL
LIN {X 0,Y 424.163,Z 521.092,A -85,B 0,C 180,E1 -9643.413,E2 -9643.413} C_VEL
LIN {X 0,Y 424.362,Z 518.576,A -85,B 0,C 180,E1 -9644.875,E2 -9644.875} C_VEL
LIN {X 0,Y 424.603,Z 515.006,A -85,B 0,C 180,E1 -9646.343,E2 -9646.343} C_VEL
LIN {X 0,Y 424.898,Z 510.264,A -85,B 0,C 180,E1 -9647.818,E2 -9647.818} C_VEL
LIN {X 0,Y 425.385,Z 504.201,A -85,B 0,C 180,E1 -9649.295,E2 -9649.295} C_VEL
LIN {X 0,Y 425.933,Z 496.58,A -85,B 0,C 180,E1 -9650.779,E2 -9650.779} C_VEL
LIN {X 0,Y 426.562,Z 488.742,A -85,B 0,C 180,E1 -9652.014,E2 -9652.014} C_VEL
LIN {X 0,Y 427.332,Z 479.105,A -85,B 0,C 180,E1 -9653.248,E2 -9653.248} C_VEL
LIN {X 0,Y 428.104,Z 468.286,A -85,B 0,C 180,E1 -9654.36,E2 -9654.36} C_VEL
LIN {X 0,Y 428.819,Z 457.794,A -85,B 0,C 180,E1 -9655.222,E2 -9655.222} C_VEL
LIN {X 0,Y 429.397,Z 446.333,A -85,B 0,C 180,E1 -9655.966,E2 -9655.966} C_VEL
LIN {X 0,Y 429.937,Z 433.311,A -85,B 0,C 180,E1 -9656.583,E2 -9656.583} C_VEL
LIN {X 0,Y 430.158,Z 420.664,A -85,B 0,C 180,E1 -9656.994,E2 -9656.994} C_VEL
LIN {X 0,Y 431.088,Z 361.581,A -85,B 0,C 180,E1 -9658.012,E2 -9658.012} C_VEL
LIN {X 0,Y 431.486,Z 331.599,A -85,B 0,C 180,E1 -9658.518,E2 -9658.518} C_VEL
LIN {X 0,Y 427.216,Z 312.312,A -85,B 0,C 180,E1 -9659.098,E2 -9659.098} C_VEL
LIN {X 0,Y 427.273,Z 307.577,A -85,B 0,C 180,E1 -9660.111,E2 -9660.111} C_VEL
LIN {X 0,Y 425.578,Z 298.851,A -85,B 0,C 180,E1 -9662.121,E2 -9662.121} C_VEL
LIN {X 0,Y 425.296,Z 297.511,A -85,B 0,C 180,E1 -9662.478,E2 -9662.478} C_VEL
LIN {X 0,Y 425.299,Z 297.507,A -85,B 0,C 180,E1 -9665.336,E2 -9665.336} C_VEL
LIN {X 0,Y 425.301,Z 297.509,A -85,B 0,C 180,E1 -9668.898,E2 -9668.898} C_VEL
LIN {X 0,Y 425.289,Z 297.508,A -85,B 0,C 180,E1 -9671.958,E2 -9671.958} C_VEL
LIN {X 0,Y 425.284,Z 297.508,A -85,B 0,C 180,E1 -9675.283,E2 -9675.283} C_VEL
LIN {X 0,Y 425.274,Z 297.513,A -85,B 0,C 180,E1 -9678.622,E2 -9678.622} C_VEL
LIN {X 0,Y 425.309,Z 297.505,A -85,B 0,C 180,E1 -9681.103,E2 -9681.103} C_VEL
LIN {X 0,Y 425.298,Z 297.506,A -85,B 0,C 180,E1 -9684.664,E2 -9684.664} C_VEL
LIN {X 0,Y 425.264,Z 297.504,A -85,B 0,C 180,E1 -9688.073,E2 -9688.073} C_VEL
LIN {X 0,Y 425.33,Z 297.499,A -85,B 0,C 180,E1 -9691.368,E2 -9691.368} C_VEL
LIN {X 0,Y 425.292,Z 297.502,A -85,B 0,C 180,E1 -9694.555,E2 -9694.555} C_VEL
LIN {X 0,Y 425.287,Z 297.508,A -85,B 0,C 180,E1 -9697.661,E2 -9697.661} C_VEL
LIN {X 0,Y 425.361,Z 297.491,A -85,B 0,C 180,E1 -9700.704,E2 -9700.704} C_VEL
LIN {X 0,Y 425.388,Z 297.494,A -85,B 0,C 180,E1 -9703.688,E2 -9703.688} C_VEL
LIN {X 0,Y 425.411,Z 297.496,A -85,B 0,C 180,E1 -9707.598,E2 -9707.598} C_VEL
LIN {X 0,Y 425.442,Z 297.49,A -85,B 0,C 180,E1 -9711.45,E2 -9711.45} C_VEL
LIN {X 0,Y 425.549,Z 297.474,A -85,B 0,C 180,E1 -9714.313,E2 -9714.313} C_VEL
LIN {X 0,Y 425.573,Z 297.47,A -85,B 0,C 180,E1 -9718.107,E2 -9718.107} C_VEL
LIN {X 0,Y 425.701,Z 297.459,A -85,B 0,C 180,E1 -9720,E2 -9720} C_VEL
LIN {X 0,Y 425.545,Z 297.469,A -85,B 0,C 180,E1 -9722.84,E2 -9722.84} C_VEL
LIN {X 0,Y 425.527,Z 297.471,A -85,B 0,C 180,E1 -9726.639,E2 -9726.639} C_VEL
LIN {X 0,Y 425.401,Z 297.49,A -85,B 0,C 180,E1 -9729.51,E2 -9729.51} C_VEL
LIN {X 0,Y 425.393,Z 297.493,A -85,B 0,C 180,E1 -9732.904,E2 -9732.904} C_VEL
LIN {X 0,Y 425.361,Z 297.497,A -85,B 0,C 180,E1 -9736.605,E2 -9736.605} C_VEL
LIN {X 0,Y 425.329,Z 297.497,A -85,B 0,C 180,E1 -9739.636,E2 -9739.636} C_VEL
LIN {X 0,Y 425.288,Z 297.507,A -85,B 0,C 180,E1 -9742.339,E2 -9742.339} C_VEL
LIN {X 0,Y 425.296,Z 297.505,A -85,B 0,C 180,E1 -9745.446,E2 -9745.446} C_VEL
LIN {X 0,Y 425.332,Z 297.501,A -85,B 0,C 180,E1 -9748.632,E2 -9748.632} C_VEL
LIN {X 0,Y 425.265,Z 297.506,A -85,B 0,C 180,E1 -9751.927,E2 -9751.927} C_VEL
LIN {X 0,Y 425.3,Z 297.505,A -85,B 0,C 180,E1 -9755.336,E2 -9755.336} C_VEL
LIN {X 0,Y 425.303,Z 297.506,A -85,B 0,C 180,E1 -9758.899,E2 -9758.899} C_VEL
LIN {X 0,Y 425.292,Z 297.505,A -85,B 0,C 180,E1 -9761.958,E2 -9761.958} C_VEL
LIN {X 0,Y 425.286,Z 297.51,A -85,B 0,C 180,E1 -9765.283,E2 -9765.283} C_VEL
LIN {X 0,Y 425.275,Z 297.508,A -85,B 0,C 180,E1 -9768.622,E2 -9768.622} C_VEL
LIN {X 0,Y 425.299,Z 297.506,A -85,B 0,C 180,E1 -9771.101,E2 -9771.101} C_VEL
LIN {X 0,Y 425.301,Z 297.505,A -85,B 0,C 180,E1 -9774.664,E2 -9774.664} C_VEL
LIN {X 0,Y 425.268,Z 297.513,A -85,B 0,C 180,E1 -9778.073,E2 -9778.073} C_VEL
LIN {X 0,Y 425.374,Z 297.499,A -85,B 0,C 180,E1 -9781.909,E2 -9781.909} C_VEL
LIN {X 0,Y 425.399,Z 297.634,A -85,B 0,C 180,E1 -9782.112,E2 -9782.112} C_VEL
LIN {X 0,Y 427.949,Z 309.635,A -85,B 0,C 180,E1 -9784.724,E2 -9784.724} C_VEL
LIN {X 0,Y 428.588,Z 314.828,A -85,B 0,C 180,E1 -9785.798,E2 -9785.798} C_VEL
LIN {X 0,Y 427.348,Z 333,A -85,B 0,C 180,E1 -9789.294,E2 -9789.294} C_VEL
LIN {X 0,Y 426.84,Z 341.856,A -85,B 0,C 180,E1 -9790.953,E2 -9790.953} C_VEL
LIN {X 0,Y 430.66,Z 364.153,A -85,B 0,C 180,E1 -9791.541,E2 -9791.541} C_VEL
LIN {X 0,Y 431.11,Z 370.054,A -85,B 0,C 180,E1 -9791.667,E2 -9791.667} C_VEL
LIN {X 0,Y 430.14,Z 450.508,A -85,B 0,C 180,E1 -9793.049,E2 -9793.049} C_VEL
LIN {X 0,Y 429.58,Z 463.626,A -85,B 0,C 180,E1 -9793.455,E2 -9793.455} C_VEL
LIN {X 0,Y 428.936,Z 476.811,A -85,B 0,C 180,E1 -9794.071,E2 -9794.071} C_VEL
LIN {X 0,Y 428.207,Z 487.913,A -85,B 0,C 180,E1 -9794.775,E2 -9794.775} C_VEL
LIN {X 0,Y 427.401,Z 499.474,A -85,B 0,C 180,E1 -9795.72,E2 -9795.72} C_VEL
LIN {X 0,Y 426.678,Z 509.896,A -85,B 0,C 180,E1 -9796.789,E2 -9796.789} C_VEL
LIN {X 0,Y 426.075,Z 518.433,A -85,B 0,C 180,E1 -9797.859,E2 -9797.859} C_VEL
LIN {X 0,Y 425.405,Z 526.325,A -85,B 0,C 180,E1 -9799.048,E2 -9799.048} C_VEL
LIN {X 0,Y 424.868,Z 534.058,A -85,B 0,C 180,E1 -9800.478,E2 -9800.478} C_VEL
LIN {X 0,Y 424.523,Z 540.278,A -85,B 0,C 180,E1 -9801.91,E2 -9801.91} C_VEL
LIN {X 0,Y 424.302,Z 545.235,A -85,B 0,C 180,E1 -9803.342,E2 -9803.342} C_VEL
LIN {X 0,Y 424.206,Z 549.073,A -85,B 0,C 180,E1 -9804.772,E2 -9804.772} C_VEL
LIN {X 0,Y 424.1,Z 551.892,A -85,B 0,C 180,E1 -9806.199,E2 -9806.199} C_VEL
LIN {X 0,Y 424.133,Z 553.231,A -85,B 0,C 180,E1 -9807.15,E2 -9807.15} C_VEL
LIN {X 0,Y 424.143,Z 554.176,A -85,B 0,C 180,E1 -9808.101,E2 -9808.101} C_VEL
LIN {X 0,Y 424.091,Z 554.725,A -85,B 0,C 180,E1 -9809.05,E2 -9809.05} C_VEL
LIN {X 0,Y 424.109,Z 554.842,A -85,B 0,C 180,E1 -9810,E2 -9810} C_VEL
LIN {X 0,Y 424.145,Z 553.903,A -85,B 0,C 180,E1 -9811.899,E2 -9811.899} C_VEL
LIN {X 0,Y 424.164,Z 552.845,A -85,B 0,C 180,E1 -9812.849,E2 -9812.849} C_VEL
LIN {X 0,Y 424.103,Z 551.328,A -85,B 0,C 180,E1 -9813.8,E2 -9813.8} C_VEL
LIN {X 0,Y 424.205,Z 548.265,A -85,B 0,C 180,E1 -9815.228,E2 -9815.228} C_VEL
LIN {X 0,Y 424.299,Z 544.131,A -85,B 0,C 180,E1 -9816.658,E2 -9816.658} C_VEL
LIN {X 0,Y 424.534,Z 537.794,A -85,B 0,C 180,E1 -9818.328,E2 -9818.328} C_VEL
LIN {X 0,Y 424.884,Z 530.887,A -85,B 0,C 180,E1 -9819.761,E2 -9819.761} C_VEL
LIN {X 0,Y 425.282,Z 523.831,A -85,B 0,C 180,E1 -9820.955,E2 -9820.955} C_VEL
LIN {X 0,Y 425.884,Z 515.332,A -85,B 0,C 180,E1 -9822.145,E2 -9822.145} C_VEL
LIN {X 0,Y 426.523,Z 504.81,A -85,B 0,C 180,E1 -9823.337,E2 -9823.337} C_VEL
LIN {X 0,Y 427.16,Z 492.946,A -85,B 0,C 180,E1 -9824.409,E2 -9824.409} C_VEL
LIN {X 0,Y 427.874,Z 481.033,A -85,B 0,C 180,E1 -9825.236,E2 -9825.236} C_VEL
LIN {X 0,Y 428.442,Z 468.615,A -85,B 0,C 180,E1 -9825.886,E2 -9825.886} C_VEL
LIN {X 0,Y 428.991,Z 455.87,A -85,B 0,C 180,E1 -9826.354,E2 -9826.354} C_VEL
LIN {X 0,Y 429.27,Z 442.452,A -85,B 0,C 180,E1 -9826.649,E2 -9826.649} C_VEL
LIN {X 0,Y 429.941,Z 366.612,A -85,B 0,C 180,E1 -9827.914,E2 -9827.914} C_VEL
LIN {X 0,Y 426.335,Z 341.855,A -85,B 0,C 180,E1 -9828.501,E2 -9828.501} C_VEL
LIN {X 0,Y 427.314,Z 323.333,A -85,B 0,C 180,E1 -9831.972,E2 -9831.972} C_VEL
LIN {X 0,Y 427.968,Z 311.362,A -85,B 0,C 180,E1 -9834.238,E2 -9834.238} C_VEL
LIN {X 0,Y 425.556,Z 298.327,A -85,B 0,C 180,E1 -9836.899,E2 -9836.899} C_VEL
LIN {X 0,Y 425.395,Z 297.497,A -85,B 0,C 180,E1 -9837.111,E2 -9837.111} C_VEL
LIN {X 0,Y 425.291,Z 297.509,A -85,B 0,C 180,E1 -9839.719,E2 -9839.719} C_VEL
LIN {X 0,Y 425.282,Z 297.505,A -85,B 0,C 180,E1 -9843.047,E2 -9843.047} C_VEL
LIN {X 0,Y 425.281,Z 297.509,A -85,B 0,C 180,E1 -9845.928,E2 -9845.928} C_VEL
LIN {X 0,Y 425.28,Z 297.506,A -85,B 0,C 180,E1 -9849.04,E2 -9849.04} C_VEL
LIN {X 0,Y 425.288,Z 297.507,A -85,B 0,C 180,E1 -9851.957,E2 -9851.957} C_VEL
LIN {X 0,Y 425.282,Z 297.505,A -85,B 0,C 180,E1 -9855.282,E2 -9855.282} C_VEL
LIN {X 0,Y 425.273,Z 297.514,A -85,B 0,C 180,E1 -9858.621,E2 -9858.621} C_VEL
LIN {X 0,Y 425.307,Z 297.505,A -85,B 0,C 180,E1 -9861.102,E2 -9861.102} C_VEL
LIN {X 0,Y 425.296,Z 297.51,A -85,B 0,C 180,E1 -9864.663,E2 -9864.663} C_VEL
LIN {X 0,Y 425.261,Z 297.508,A -85,B 0,C 180,E1 -9868.072,E2 -9868.072} C_VEL
LIN {X 0,Y 425.327,Z 297.502,A -85,B 0,C 180,E1 -9871.367,E2 -9871.367} C_VEL
LIN {X 0,Y 425.291,Z 297.506,A -85,B 0,C 180,E1 -9874.554,E2 -9874.554} C_VEL
LIN {X 0,Y 425.284,Z 297.507,A -85,B 0,C 180,E1 -9877.661,E2 -9877.661} C_VEL
LIN {X 0,Y 425.358,Z 297.498,A -85,B 0,C 180,E1 -9880.704,E2 -9880.704} C_VEL
LIN {X 0,Y 425.384,Z 297.495,A -85,B 0,C 180,E1 -9883.688,E2 -9883.688} C_VEL
LIN {X 0,Y 425.407,Z 297.495,A -85,B 0,C 180,E1 -9887.598,E2 -9887.598} C_VEL
LIN {X 0,Y 425.438,Z 297.493,A -85,B 0,C 180,E1 -9891.45,E2 -9891.45} C_VEL
LIN {X 0,Y 425.547,Z 297.473,A -85,B 0,C 180,E1 -9894.313,E2 -9894.313} C_VEL
LIN {X 0,Y 425.567,Z 297.472,A -85,B 0,C 180,E1 -9898.107,E2 -9898.107} C_VEL
LIN {X 0,Y 425.695,Z 297.458,A -85,B 0,C 180,E1 -9900,E2 -9900} C_VEL
LIN {X 0,Y 425.541,Z 297.473,A -85,B 0,C 180,E1 -9902.84,E2 -9902.84} C_VEL
LIN {X 0,Y 425.492,Z 297.479,A -85,B 0,C 180,E1 -9906.521,E2 -9906.521} C_VEL
LIN {X 0,Y 425.395,Z 297.493,A -85,B 0,C 180,E1 -9909.509,E2 -9909.509} C_VEL
LIN {X 0,Y 425.388,Z 297.492,A -85,B 0,C 180,E1 -9912.904,E2 -9912.904} C_VEL
LIN {X 0,Y 425.355,Z 297.499,A -85,B 0,C 180,E1 -9916.605,E2 -9916.605} C_VEL
LIN {X 0,Y 425.322,Z 297.501,A -85,B 0,C 180,E1 -9919.636,E2 -9919.636} C_VEL
LIN {X 0,Y 425.282,Z 297.513,A -85,B 0,C 180,E1 -9922.339,E2 -9922.339} C_VEL
LIN {X 0,Y 425.315,Z 297.506,A -85,B 0,C 180,E1 -9924.658,E2 -9924.658} C_VEL
LIN {X 0,Y 425.34,Z 297.498,A -85,B 0,C 180,E1 -9927.558,E2 -9927.558} C_VEL
LIN {X 0,Y 425.282,Z 297.51,A -85,B 0,C 180,E1 -9930.816,E2 -9930.816} C_VEL
LIN {X 0,Y 425.306,Z 297.505,A -85,B 0,C 180,E1 -9934.288,E2 -9934.288} C_VEL
LIN {X 0,Y 425.273,Z 297.506,A -85,B 0,C 180,E1 -9937.695,E2 -9937.695} C_VEL
LIN {X 0,Y 425.275,Z 297.51,A -85,B 0,C 180,E1 -9940.521,E2 -9940.521} C_VEL
LIN {X 0,Y 425.253,Z 297.511,A -85,B 0,C 180,E1 -9943.351,E2 -9943.351} C_VEL
LIN {X 0,Y 425.253,Z 297.509,A -85,B 0,C 180,E1 -9946.044,E2 -9946.044} C_VEL
LIN {X 0,Y 425.25,Z 297.512,A -85,B 0,C 180,E1 -9949.484,E2 -9949.484} C_VEL
LIN {X 0,Y 425.273,Z 297.507,A -85,B 0,C 180,E1 -9952.489,E2 -9952.489} C_VEL
LIN {X 0,Y 425.302,Z 297.504,A -85,B 0,C 180,E1 -9955.818,E2 -9955.818} C_VEL
LIN {X 0,Y 425.287,Z 297.511,A -85,B 0,C 180,E1 -9959.24,E2 -9959.24} C_VEL
LIN {X 0,Y 425.302,Z 297.511,A -85,B 0,C 180,E1 -9961.366,E2 -9961.366} C_VEL
LIN {X 0,Y 425.255,Z 297.508,A -85,B 0,C 180,E1 -9964.553,E2 -9964.553} C_VEL
LIN {X 0,Y 425.29,Z 297.51,A -85,B 0,C 180,E1 -9967.73,E2 -9967.73} C_VEL
LIN {X 0,Y 425.359,Z 297.496,A -85,B 0,C 180,E1 -9970.704,E2 -9970.704} C_VEL
LIN {X 0,Y 425.386,Z 297.5,A -85,B 0,C 180,E1 -9973.689,E2 -9973.689} C_VEL
LIN {X 0,Y 425.407,Z 297.497,A -85,B 0,C 180,E1 -9977.599,E2 -9977.599} C_VEL
LIN {X 0,Y 425.391,Z 297.565,A -85,B 0,C 180,E1 -9978.384,E2 -9978.384} C_VEL
LIN {X 0,Y 426.78,Z 306.031,A -85,B 0,C 180,E1 -9980.283,E2 -9980.283} C_VEL
LIN {X 0,Y 426.711,Z 312.531,A -85,B 0,C 180,E1 -9981.619,E2 -9981.619} C_VEL
LIN {X 0,Y 430.222,Z 331.666,A -85,B 0,C 180,E1 -9982.083,E2 -9982.083} C_VEL
LIN {X 0,Y 429.241,Z 419.556,A -85,B 0,C 180,E1 -9983.567,E2 -9983.567} C_VEL
LIN {X 0,Y 429.1,Z 426.036,A -85,B 0,C 180,E1 -9983.744,E2 -9983.744} C_VEL
LIN {X 0,Y 427.743,Z 433.602,A -85,B 0,C 180,E1 -9983.971,E2 -9983.971} C_VEL
LIN {X 0,Y 425.118,Z 440.899,A -85,B 0,C 180,E1 -9984.21,E2 -9984.21} C_VEL
LIN {X 0,Y 422.083,Z 449.879,A -85,B 0,C 180,E1 -9984.616,E2 -9984.616} C_VEL
LIN {X 0,Y 421.232,Z 455.15,A -85,B 0,C 180,E1 -9984.942,E2 -9984.942} C_VEL
LIN {X 0,Y 420.45,Z 466.265,A -85,B 0,C 180,E1 -9985.807,E2 -9985.807} C_VEL
LIN {X 0,Y 419.734,Z 477.081,A -85,B 0,C 180,E1 -9986.881,E2 -9986.881} C_VEL
LIN {X 0,Y 419.081,Z 486.784,A -85,B 0,C 180,E1 -9988.078,E2 -9988.078} C_VEL
LIN {X 0,Y 418.596,Z 494.738,A -85,B 0,C 180,E1 -9989.279,E2 -9989.279} C_VEL
LIN {X 0,Y 418.035,Z 502.571,A -85,B 0,C 180,E1 -9990.723,E2 -9990.723} C_VEL
LIN {X 0,Y 417.696,Z 507.876,A -85,B 0,C 180,E1 -9991.929,E2 -9991.929} C_VEL
LIN {X 0,Y 417.46,Z 513.068,A -85,B 0,C 180,E1 -9993.378,E2 -9993.378} C_VEL
LIN {X 0,Y 417.245,Z 517.115,A -85,B 0,C 180,E1 -9994.831,E2 -9994.831} C_VEL
LIN {X 0,Y 417.246,Z 520.304,A -85,B 0,C 180,E1 -9996.394,E2 -9996.394} C_VEL
LIN {X 0,Y 417.038,Z 522.156,A -85,B 0,C 180,E1 -9997.748,E2 -9997.748} C_VEL
LIN {X 0,Y 416.971,Z 523.025,A -85,B 0,C 180,E1 -9998.725,E2 -9998.725} C_VEL
LIN {X 0,Y 416.991,Z 523.486,A -85,B 0,C 180,E1 -10000.684,E2 -10000.684} C_VEL
LIN {X 0,Y 417.072,Z 522.738,A -85,B 0,C 180,E1 -10002.22,E2 -10002.22} C_VEL
LIN {X 0,Y 417.09,Z 521.157,A -85,B 0,C 180,E1 -10003.645,E2 -10003.645} C_VEL
LIN {X 0,Y 417.348,Z 518.546,A -85,B 0,C 180,E1 -10005.13,E2 -10005.13} C_VEL
LIN {X 0,Y 417.583,Z 514.876,A -85,B 0,C 180,E1 -10006.626,E2 -10006.626} C_VEL
LIN {X 0,Y 417.92,Z 510.026,A -85,B 0,C 180,E1 -10008.126,E2 -10008.126} C_VEL
LIN {X 0,Y 418.443,Z 503.844,A -85,B 0,C 180,E1 -10009.628,E2 -10009.628} C_VEL
LIN {X 0,Y 419.072,Z 496.088,A -85,B 0,C 180,E1 -10011.135,E2 -10011.135} C_VEL
LIN {X 0,Y 419.77,Z 488.066,A -85,B 0,C 180,E1 -10012.389,E2 -10012.389} C_VEL
LIN {X 0,Y 420.577,Z 478.182,A -85,B 0,C 180,E1 -10013.644,E2 -10013.644} C_VEL
LIN {X 0,Y 421.439,Z 467.124,A -85,B 0,C 180,E1 -10014.771,E2 -10014.771} C_VEL
LIN {X 0,Y 422.147,Z 456.225,A -85,B 0,C 180,E1 -10015.649,E2 -10015.649} C_VEL
LIN {X 0,Y 422.777,Z 445.177,A -85,B 0,C 180,E1 -10016.344,E2 -10016.344} C_VEL
LIN {X 0,Y 423.239,Z 432.551,A -85,B 0,C 180,E1 -10016.937,E2 -10016.937} C_VEL
LIN {X 0,Y 423.507,Z 420.623,A -85,B 0,C 180,E1 -10017.319,E2 -10017.319} C_VEL
LIN {X 0,Y 424.824,Z 332.4,A -85,B 0,C 180,E1 -10018.853,E2 -10018.853} C_VEL
LIN {X 0,Y 420.418,Z 312.608,A -85,B 0,C 180,E1 -10019.457,E2 -10019.457} C_VEL
LIN {X 0,Y 420.3,Z 308.395,A -85,B 0,C 180,E1 -10020.386,E2 -10020.386} C_VEL
LIN {X 0,Y 418.242,Z 298.389,A -85,B 0,C 180,E1 -10022.755,E2 -10022.755} C_VEL
LIN {X 0,Y 418.243,Z 298.39,A -85,B 0,C 180,E1 -10026.024,E2 -10026.024} C_VEL
LIN {X 0,Y 418.246,Z 298.386,A -85,B 0,C 180,E1 -10029.683,E2 -10029.683} C_VEL
LIN {X 0,Y 418.229,Z 298.388,A -85,B 0,C 180,E1 -10032.321,E2 -10032.321} C_VEL
LIN {X 0,Y 418.235,Z 298.388,A -85,B 0,C 180,E1 -10035.109,E2 -10035.109} C_VEL
LIN {X 0,Y 418.239,Z 298.384,A -85,B 0,C 180,E1 -10037.767,E2 -10037.767} C_VEL
LIN {X 0,Y 418.255,Z 298.385,A -85,B 0,C 180,E1 -10040.619,E2 -10040.619} C_VEL
LIN {X 0,Y 418.242,Z 298.381,A -85,B 0,C 180,E1 -10043.976,E2 -10043.976} C_VEL
LIN {X 0,Y 418.257,Z 298.383,A -85,B 0,C 180,E1 -10047.156,E2 -10047.156} C_VEL
LIN {X 0,Y 418.268,Z 298.38,A -85,B 0,C 180,E1 -10050.896,E2 -10050.896} C_VEL
LIN {X 0,Y 418.268,Z 298.377,A -85,B 0,C 180,E1 -10054.096,E2 -10054.096} C_VEL
LIN {X 0,Y 418.231,Z 298.383,A -85,B 0,C 180,E1 -10057.264,E2 -10057.264} C_VEL
LIN {X 0,Y 418.282,Z 298.372,A -85,B 0,C 180,E1 -10060.364,E2 -10060.364} C_VEL
LIN {X 0,Y 418.316,Z 298.38,A -85,B 0,C 180,E1 -10063.405,E2 -10063.405} C_VEL
LIN {X 0,Y 418.346,Z 298.371,A -85,B 0,C 180,E1 -10067,E2 -10067} C_VEL
LIN {X 0,Y 418.34,Z 298.372,A -85,B 0,C 180,E1 -10070.329,E2 -10070.329} C_VEL
LIN {X 0,Y 418.513,Z 298.349,A -85,B 0,C 180,E1 -10072.28,E2 -10072.28} C_VEL
LIN {X 0,Y 418.509,Z 298.352,A -85,B 0,C 180,E1 -10074.217,E2 -10074.217} C_VEL
LIN {X 0,Y 418.542,Z 298.345,A -85,B 0,C 180,E1 -10078.076,E2 -10078.076} C_VEL
LIN {X 0,Y 418.67,Z 298.334,A -85,B 0,C 180,E1 -10080,E2 -10080} C_VEL
